LIN {X 0.080,Y -429.880,Z 672.901,A 0.000,B 0.000,C 90.000,E1 18.181} C_DIS
LIN {X -0.115,Y -431.372,Z 672.890,A 0.000,B 0.000,C 90.000,E1 16.205} C_DIS
LIN {X -0.059,Y -433.748,Z 672.875,A 0.000,B 0.000,C 90.000,E1 13.536} C_DIS
LIN {X 0.029,Y -435.804,Z 672.864,A 0.000,B 0.000,C 90.000,E1 11.535} C_DIS
LIN {X 0.134,Y -438.251,Z 672.851,A 0.000,B 0.000,C 90.000,E1 9.208} C_DIS
LIN {X -0.200,Y -440.989,Z 672.839,A 0.000,B 0.000,C 90.000,E1 6.947} C_DIS
LIN {X 0.152,Y -443.481,Z 672.828,A 0.000,B 0.000,C 90.000,E1 4.935} C_DIS
LIN {X -0.046,Y -447.163,Z 672.813,A 0.000,B 0.000,C 90.000,E1 2.350} C_DIS
LIN {X -0.119,Y -451.557,Z 672.797,A 0.000,B 0.000,C 90.000,E1 359.484} C_DIS
LIN {X 0.170,Y -455.546,Z 672.785,A 0.000,B 0.000,C 90.000,E1 357.192} C_DIS
LIN {X 0.214,Y -458.466,Z 672.776,A 0.000,B 0.000,C 90.000,E1 355.584} C_DIS
LIN {X -0.148,Y -461.460,Z 672.767,A 0.000,B 0.000,C 90.000,E1 354.033} C_DIS
LIN {X 0.093,Y -465.598,Z 672.754,A 0.000,B 0.000,C 90.000,E1 351.781} C_DIS
LIN {X -0.140,Y -469.084,Z 672.744,A 0.000,B 0.000,C 90.000,E1 349.916} C_DIS
LIN {X 0.174,Y -472.431,Z 672.733,A 0.000,B 0.000,C 90.000,E1 347.993} C_DIS
LIN {X 0.025,Y -476.365,Z 672.721,A 0.000,B 0.000,C 90.000,E1 345.825} C_DIS
LIN {X -0.099,Y -479.865,Z 672.711,A 0.000,B 0.000,C 90.000,E1 343.976} C_DIS
LIN {X -0.142,Y -483.419,Z 672.701,A 0.000,B 0.000,C 90.000,E1 342.127} C_DIS
LIN {X 0.212,Y -487.775,Z 672.689,A 0.000,B 0.000,C 90.000,E1 339.934} C_DIS
LIN {X 0.229,Y -492.077,Z 672.677,A 0.000,B 0.000,C 90.000,E1 337.794} C_DIS
LIN {X -0.025,Y -494.971,Z 672.668,A 0.000,B 0.000,C 90.000,E1 336.305} C_DIS
LIN {X -0.028,Y -497.759,Z 672.660,A 0.000,B 0.000,C 90.000,E1 334.793} C_DIS
LIN {X 0.240,Y -500.778,Z 672.652,A 0.000,B 0.000,C 90.000,E1 333.256} C_DIS
LIN {X -0.147,Y -501.596,Z 672.650,A 0.000,B 0.000,C 90.000,E1 332.999} C_DIS
LIN {X 0.034,Y -502.535,Z 672.648,A 0.000,B 0.000,C 90.000,E1 332.692} C_DIS
LIN {X -0.118,Y -503.291,Z 672.647,A 0.000,B 0.000,C 90.000,E1 332.410} C_DIS
LIN {X 0.254,Y -505.894,Z 672.643,A 0.000,B 0.000,C 90.000,E1 331.769} C_DIS
LIN {X 0.141,Y -507.043,Z 672.642,A 0.000,B 0.000,C 90.000,E1 331.591} C_DIS
LIN {X 0.151,Y -510.292,Z 672.640,A 0.000,B 0.000,C 90.000,E1 331.179} C_DIS
LIN {X 0.180,Y -513.746,Z 672.638,A 0.000,B 0.000,C 90.000,E1 330.845} C_DIS
LIN {X 0.160,Y -516.813,Z 672.637,A 0.000,B 0.000,C 90.000,E1 330.589} C_DIS
LIN {X 0.046,Y -533.052,Z 672.630,A 0.000,B 0.000,C 90.000,E1 329.459} C_DIS
LIN {X -0.033,Y -540.415,Z 672.627,A 0.000,B 0.000,C 90.000,E1 328.918} C_DIS
LIN {X -0.038,Y -546.271,Z 672.625,A 0.000,B 0.000,C 90.000,E1 328.456} C_DIS
LIN {X -0.173,Y -551.951,Z 672.622,A 0.000,B 0.000,C 90.000,E1 327.995} C_DIS
LIN {X -0.024,Y -560.113,Z 672.618,A 0.000,B 0.000,C 90.000,E1 327.248} C_DIS
LIN {X -0.061,Y -569.208,Z 672.613,A 0.000,B 0.000,C 90.000,E1 326.373} C_DIS
LIN {X -0.056,Y -578.305,Z 672.608,A 0.000,B 0.000,C 90.000,E1 325.468} C_DIS
LIN {X 0.240,Y -588.531,Z 672.602,A 0.000,B 0.000,C 90.000,E1 324.402} C_DIS
LIN {X -0.015,Y -593.457,Z 672.600,A 0.000,B 0.000,C 90.000,E1 323.909} C_DIS
LIN {X 0.212,Y -600.526,Z 672.595,A 0.000,B 0.000,C 90.000,E1 323.130} C_DIS
LIN {X 0.309,Y -606.223,Z 672.592,A 0.000,B 0.000,C 90.000,E1 322.477} C_DIS
LIN {X 0.322,Y -611.798,Z 672.588,A 0.000,B 0.000,C 90.000,E1 321.823} C_DIS
LIN {X -0.183,Y -618.774,Z 672.583,A 0.000,B 0.000,C 90.000,E1 320.964} C_DIS
LIN {X 0.324,Y -623.427,Z 672.580,A 0.000,B 0.000,C 90.000,E1 320.275} C_DIS
LIN {X 0.001,Y -627.856,Z 672.576,A 0.000,B 0.000,C 90.000,E1 319.666} C_DIS
LIN {X -0.318,Y -632.855,Z 672.572,A 0.000,B 0.000,C 90.000,E1 318.933} C_DIS
LIN {X -0.175,Y -637.627,Z 672.568,A 0.000,B 0.000,C 90.000,E1 318.162} C_DIS
LIN {X -0.006,Y -642.937,Z 672.563,A 0.000,B 0.000,C 90.000,E1 317.268} C_DIS
LIN {X -0.301,Y -648.669,Z 672.557,A 0.000,B 0.000,C 90.000,E1 316.296} C_DIS
LIN {X -0.051,Y -654.087,Z 672.552,A 0.000,B 0.000,C 90.000,E1 315.283} C_DIS
LIN {X -0.180,Y -658.514,Z 672.547,A 0.000,B 0.000,C 90.000,E1 314.433} C_DIS
LIN {X 0.187,Y -663.844,Z 672.541,A 0.000,B 0.000,C 90.000,E1 313.299} C_DIS
LIN {X -0.302,Y -668.345,Z 672.535,A 0.000,B 0.000,C 90.000,E1 312.366} C_DIS
LIN {X 0.201,Y -671.663,Z 672.531,A 0.000,B 0.000,C 90.000,E1 311.595} C_DIS
LIN {X -0.103,Y -676.763,Z 672.525,A 0.000,B 0.000,C 90.000,E1 310.415} C_DIS
LIN {X -0.034,Y -679.526,Z 672.521,A 0.000,B 0.000,C 90.000,E1 309.688} C_DIS
LIN {X 0.113,Y -681.274,Z 672.518,A 0.000,B 0.000,C 90.000,E1 309.197} C_DIS
LIN {X -0.041,Y -685.072,Z 672.511,A 0.000,B 0.000,C 90.000,E1 308.016} C_DIS
LIN {X -0.223,Y -687.170,Z 672.507,A 0.000,B 0.000,C 90.000,E1 307.317} C_DIS
LIN {X -0.337,Y -689.640,Z 672.502,A 0.000,B 0.000,C 90.000,E1 306.377} C_DIS
LIN {X 0.137,Y -691.969,Z 672.497,A 0.000,B 0.000,C 90.000,E1 305.391} C_DIS
LIN {X 0.070,Y -694.004,Z 672.491,A 0.000,B 0.000,C 90.000,E1 304.452} C_DIS
LIN {X 0.203,Y -695.870,Z 672.486,A 0.000,B 0.000,C 90.000,E1 303.499} C_DIS
LIN {X 0.366,Y -697.540,Z 672.481,A 0.000,B 0.000,C 90.000,E1 302.546} C_DIS
LIN {X 0.206,Y -699.243,Z 672.474,A 0.000,B 0.000,C 90.000,E1 301.386} C_DIS
LIN {X 0.045,Y -700.466,Z 672.469,A 0.000,B 0.000,C 90.000,E1 300.463} C_DIS
LIN {X -0.097,Y -701.424,Z 672.464,A 0.000,B 0.000,C 90.000,E1 299.539} C_DIS
LIN {X 0.048,Y -702.476,Z 672.458,A 0.000,B 0.000,C 90.000,E1 298.359} C_DIS
LIN {X -0.179,Y -703.813,Z 672.449,A 0.000,B 0.000,C 90.000,E1 296.744} C_DIS
LIN {X 0.021,Y -704.458,Z 672.443,A 0.000,B 0.000,C 90.000,E1 295.796} C_DIS
LIN {X -0.327,Y -704.513,Z 672.442,A 0.000,B 0.000,C 90.000,E1 295.591} C_DIS
LIN {X 0.245,Y -704.053,Z 672.440,A 0.000,B 0.000,C 90.000,E1 295.079} C_DIS
LIN {X -0.406,Y -703.556,Z 672.438,A 0.000,B 0.000,C 90.000,E1 294.899} C_DIS
LIN {X 0.159,Y -701.504,Z 672.436,A 0.000,B 0.000,C 90.000,E1 294.387} C_DIS
LIN {X 0.297,Y -700.902,Z 672.435,A 0.000,B 0.000,C 90.000,E1 294.259} C_DIS
LIN {X 0.148,Y -699.998,Z 672.434,A 0.000,B 0.000,C 90.000,E1 294.155} C_DIS
LIN {X -0.354,Y -698.653,Z 672.434,A 0.000,B 0.000,C 90.000,E1 294.079} C_DIS
LIN {X -0.100,Y -692.661,Z 672.431,A 0.000,B 0.000,C 90.000,E1 293.643} C_DIS
LIN {X 0.271,Y -690.364,Z 672.431,A 0.000,B 0.000,C 90.000,E1 293.515} C_DIS
LIN {X 0.067,Y -688.120,Z 672.430,A 0.000,B 0.000,C 90.000,E1 293.462} C_DIS
LIN {X 0.247,Y -679.913,Z 672.429,A 0.000,B 0.000,C 90.000,E1 293.259} C_DIS
LIN {X 0.214,Y -670.677,Z 672.429,A 0.000,B 0.000,C 90.000,E1 293.153} C_DIS
LIN {X -0.217,Y -665.106,Z 672.428,A 0.000,B 0.000,C 90.000,E1 293.131} C_DIS
LIN {X 0.275,Y -655.083,Z 672.428,A 0.000,B 0.000,C 90.000,E1 292.950} C_DIS
LIN {X -0.154,Y -645.323,Z 672.427,A 0.000,B 0.000,C 90.000,E1 292.823} C_DIS
LIN {X 0.209,Y -635.120,Z 672.426,A 0.000,B 0.000,C 90.000,E1 292.589} C_DIS
LIN {X 0.133,Y -621.781,Z 672.424,A 0.000,B 0.000,C 90.000,E1 292.280} C_DIS
LIN {X -0.232,Y -604.948,Z 672.421,A 0.000,B 0.000,C 90.000,E1 291.844} C_DIS
LIN {X -0.161,Y -577.296,Z 672.416,A 0.000,B 0.000,C 90.000,E1 290.972} C_DIS
LIN {X -0.053,Y -563.094,Z 672.414,A 0.000,B 0.000,C 90.000,E1 290.556} C_DIS
LIN {X -0.047,Y -556.572,Z 672.413,A 0.000,B 0.000,C 90.000,E1 290.248} C_DIS
LIN {X -0.095,Y -556.479,Z 672.412,A 0.000,B 0.000,C 90.000,E1 290.248} C_DIS
LIN {X 0.094,Y -555.287,Z 672.412,A 0.000,B 0.000,C 90.000,E1 290.066} C_DIS
LIN {X 0.052,Y -555.271,Z 672.412,A 0.000,B 0.000,C 90.000,E1 290.066} C_DIS
LIN {X 0.022,Y -554.576,Z 672.410,A 0.000,B 0.000,C 90.000,E1 289.704} C_DIS
LIN {X 0.188,Y -554.054,Z 672.399,A 0.000,B 0.000,C 90.000,E1 287.873} C_DIS
LIN {X -0.264,Y -553.758,Z 672.393,A 0.000,B 0.000,C 90.000,E1 286.804} C_DIS
LIN {X -0.328,Y -553.213,Z 672.384,A 0.000,B 0.000,C 90.000,E1 285.134} C_DIS
LIN {X 0.001,Y -552.630,Z 672.376,A 0.000,B 0.000,C 90.000,E1 283.703} C_DIS
LIN {X 0.054,Y -551.874,Z 672.368,A 0.000,B 0.000,C 90.000,E1 282.299} C_DIS
LIN {X 0.215,Y -551.004,Z 672.359,A 0.000,B 0.000,C 90.000,E1 280.602} C_DIS
LIN {X -0.182,Y -550.230,Z 672.348,A 0.000,B 0.000,C 90.000,E1 278.681} C_DIS
LIN {X 0.195,Y -549.869,Z 672.340,A 0.000,B 0.000,C 90.000,E1 277.239} C_DIS
LIN {X 0.024,Y -549.613,Z 672.333,A 0.000,B 0.000,C 90.000,E1 275.853} C_DIS
LIN {X -0.029,Y -549.376,Z 672.320,A 0.000,B 0.000,C 90.000,E1 273.612} C_DIS
LIN {X 0.252,Y -549.149,Z 672.312,A 0.000,B 0.000,C 90.000,E1 272.178} C_DIS
LIN {X -0.074,Y -548.777,Z 672.306,A 0.000,B 0.000,C 90.000,E1 271.088} C_DIS
LIN {X 0.180,Y -548.088,Z 672.298,A 0.000,B 0.000,C 90.000,E1 269.656} C_DIS
LIN {X -0.130,Y -547.287,Z 672.290,A 0.000,B 0.000,C 90.000,E1 268.282} C_DIS
LIN {X 0.173,Y -546.280,Z 672.281,A 0.000,B 0.000,C 90.000,E1 266.560} C_DIS
LIN {X -0.115,Y -545.287,Z 672.273,A 0.000,B 0.000,C 90.000,E1 265.179} C_DIS
LIN {X 0.120,Y -544.116,Z 672.265,A 0.000,B 0.000,C 90.000,E1 263.742} C_DIS
LIN {X -0.232,Y -543.078,Z 672.259,A 0.000,B 0.000,C 90.000,E1 262.648} C_DIS
LIN {X 0.163,Y -541.204,Z 672.250,A 0.000,B 0.000,C 90.000,E1 260.905} C_DIS
LIN {X 0.140,Y -539.088,Z 672.237,A 0.000,B 0.000,C 90.000,E1 258.634} C_DIS
LIN {X 0.209,Y -536.968,Z 672.223,A 0.000,B 0.000,C 90.000,E1 256.061} C_DIS
LIN {X 0.240,Y -535.696,Z 672.215,A 0.000,B 0.000,C 90.000,E1 254.629} C_DIS
LIN {X 0.063,Y -534.559,Z 672.208,A 0.000,B 0.000,C 90.000,E1 253.504} C_DIS
LIN {X -0.044,Y -532.250,Z 672.196,A 0.000,B 0.000,C 90.000,E1 251.221} C_DIS
LIN {X -0.143,Y -531.429,Z 672.191,A 0.000,B 0.000,C 90.000,E1 250.369} C_DIS
LIN {X -0.061,Y -529.990,Z 672.185,A 0.000,B 0.000,C 90.000,E1 249.209} C_DIS
LIN {X -0.133,Y -527.570,Z 672.175,A 0.000,B 0.000,C 90.000,E1 247.486} C_DIS
LIN {X 0.084,Y -525.904,Z 672.168,A 0.000,B 0.000,C 90.000,E1 246.305} C_DIS
LIN {X -0.141,Y -522.911,Z 672.159,A 0.000,B 0.000,C 90.000,E1 244.588} C_DIS
LIN {X 0.222,Y -520.768,Z 672.152,A 0.000,B 0.000,C 90.000,E1 243.384} C_DIS
LIN {X 0.119,Y -517.300,Z 672.143,A 0.000,B 0.000,C 90.000,E1 241.641} C_DIS
LIN {X 0.171,Y -514.866,Z 672.136,A 0.000,B 0.000,C 90.000,E1 240.461} C_DIS
LIN {X 0.090,Y -511.648,Z 672.128,A 0.000,B 0.000,C 90.000,E1 238.997} C_DIS
LIN {X -0.052,Y -508.421,Z 672.120,A 0.000,B 0.000,C 90.000,E1 237.533} C_DIS
LIN {X 0.289,Y -505.035,Z 672.111,A 0.000,B 0.000,C 90.000,E1 236.008} C_DIS
LIN {X -0.019,Y -502.131,Z 672.105,A 0.000,B 0.000,C 90.000,E1 234.848} C_DIS
LIN {X -0.039,Y -497.638,Z 672.095,A 0.000,B 0.000,C 90.000,E1 233.050} C_DIS
LIN {X 0.010,Y -492.473,Z 672.083,A 0.000,B 0.000,C 90.000,E1 230.928} C_DIS
LIN {X 0.091,Y -489.603,Z 672.076,A 0.000,B 0.000,C 90.000,E1 229.703} C_DIS
LIN {X 0.210,Y -485.948,Z 672.068,A 0.000,B 0.000,C 90.000,E1 228.162} C_DIS
LIN {X -0.026,Y -480.144,Z 672.054,A 0.000,B 0.000,C 90.000,E1 225.729} C_DIS
LIN {X 0.013,Y -475.706,Z 672.044,A 0.000,B 0.000,C 90.000,E1 223.866} C_DIS
LIN {X -0.031,Y -471.424,Z 672.033,A 0.000,B 0.000,C 90.000,E1 222.000} C_DIS
LIN {X 0.002,Y -466.055,Z 672.019,A 0.000,B 0.000,C 90.000,E1 219.483} C_DIS
LIN {X 0.101,Y -462.792,Z 672.011,A 0.000,B 0.000,C 90.000,E1 217.890} C_DIS
LIN {X -0.009,Y -458.282,Z 671.998,A 0.000,B 0.000,C 90.000,E1 215.678} C_DIS
LIN {X -0.230,Y -454.694,Z 671.988,A 0.000,B 0.000,C 90.000,E1 213.785} C_DIS
LIN {X 0.213,Y -451.026,Z 671.977,A 0.000,B 0.000,C 90.000,E1 211.799} C_DIS
LIN {X 0.167,Y -446.761,Z 671.964,A 0.000,B 0.000,C 90.000,E1 209.539} C_DIS
LIN {X 0.176,Y -442.726,Z 671.952,A 0.000,B 0.000,C 90.000,E1 207.257} C_DIS
LIN {X -0.010,Y -439.755,Z 671.943,A 0.000,B 0.000,C 90.000,E1 205.643} C_DIS
LIN {X 0.017,Y -435.666,Z 671.930,A 0.000,B 0.000,C 90.000,E1 203.334} C_DIS
LIN {X -0.047,Y -432.011,Z 671.919,A 0.000,B 0.000,C 90.000,E1 201.354} C_DIS
LIN {X 0.196,Y -428.409,Z 671.908,A 0.000,B 0.000,C 90.000,E1 199.322} C_DIS
LIN {X -0.090,Y -423.799,Z 671.893,A 0.000,B 0.000,C 90.000,E1 196.677} C_DIS
LIN {X 0.180,Y -420.959,Z 671.883,A 0.000,B 0.000,C 90.000,E1 194.954} C_DIS
LIN {X -0.178,Y -418.673,Z 671.876,A 0.000,B 0.000,C 90.000,E1 193.647} C_DIS
LIN {X 0.068,Y -413.636,Z 671.859,A 0.000,B 0.000,C 90.000,E1 190.546} C_DIS
LIN {X -0.136,Y -411.008,Z 671.849,A 0.000,B 0.000,C 90.000,E1 188.859} C_DIS
LIN {X -0.028,Y -407.872,Z 671.838,A 0.000,B 0.000,C 90.000,E1 186.777} C_DIS
LIN {X -0.120,Y -403.635,Z 671.820,A 0.000,B 0.000,C 90.000,E1 183.669} C_DIS
LIN {X 0.094,Y -401.103,Z 671.809,A 0.000,B 0.000,C 90.000,E1 181.547} C_DIS
LIN {X 0.125,Y -398.349,Z 671.793,A 0.000,B 0.000,C 90.000,E1 178.740} C_DIS
LIN {X -0.061,Y -395.440,Z 671.772,A 0.000,B 0.000,C 90.000,E1 174.894} C_DIS
LIN {X -0.008,Y -394.198,Z 671.758,A 0.000,B 0.000,C 90.000,E1 172.413} C_DIS
LIN {X 0.097,Y -393.498,Z 671.746,A 0.000,B 0.000,C 90.000,E1 170.274} C_DIS
LIN {X -0.076,Y -393.038,Z 671.734,A 0.000,B 0.000,C 90.000,E1 168.173} C_DIS
LIN {X -0.083,Y -392.879,Z 671.722,A 0.000,B 0.000,C 90.000,E1 166.047} C_DIS
LIN {X 0.010,Y -392.836,Z 671.707,A 0.000,B 0.000,C 90.000,E1 163.196} C_DIS
LIN {X -0.109,Y -392.982,Z 671.693,A 0.000,B 0.000,C 90.000,E1 160.732} C_DIS
LIN {X -0.078,Y -393.142,Z 671.683,A 0.000,B 0.000,C 90.000,E1 158.954} C_DIS
LIN {X 0.155,Y -393.420,Z 671.671,A 0.000,B 0.000,C 90.000,E1 156.794} C_DIS
LIN {X -0.175,Y -393.732,Z 671.659,A 0.000,B 0.000,C 90.000,E1 154.717} C_DIS
LIN {X 0.018,Y -394.135,Z 671.648,A 0.000,B 0.000,C 90.000,E1 152.564} C_DIS
LIN {X 0.018,Y -394.563,Z 671.638,A 0.000,B 0.000,C 90.000,E1 150.795} C_DIS
LIN {X 0.227,Y -394.992,Z 671.628,A 0.000,B 0.000,C 90.000,E1 148.997} C_DIS
LIN {X -0.024,Y -395.679,Z 671.616,A 0.000,B 0.000,C 90.000,E1 146.914} C_DIS
LIN {X 0.227,Y -397.116,Z 671.599,A 0.000,B 0.000,C 90.000,E1 143.703} C_DIS
LIN {X -0.050,Y -398.754,Z 671.583,A 0.000,B 0.000,C 90.000,E1 140.928} C_DIS
LIN {X -0.142,Y -400.412,Z 671.569,A 0.000,B 0.000,C 90.000,E1 138.485} C_DIS
LIN {X -0.018,Y -401.423,Z 671.562,A 0.000,B 0.000,C 90.000,E1 137.067} C_DIS
LIN {X -0.222,Y -402.976,Z 671.550,A 0.000,B 0.000,C 90.000,E1 135.000} C_DIS
LIN {X -0.172,Y -404.024,Z 671.544,A 0.000,B 0.000,C 90.000,E1 133.947} C_DIS
LIN {X -0.050,Y -404.439,Z 671.542,A 0.000,B 0.000,C 90.000,E1 133.581} C_DIS
LIN {X 0.102,Y -406.028,Z 671.537,A 0.000,B 0.000,C 90.000,E1 132.690} C_DIS
LIN {X 0.018,Y -406.708,Z 671.536,A 0.000,B 0.000,C 90.000,E1 132.528} C_DIS
LIN {X 0.114,Y -408.061,Z 671.534,A 0.000,B 0.000,C 90.000,E1 132.081} C_DIS
LIN {X -0.167,Y -411.535,Z 671.531,A 0.000,B 0.000,C 90.000,E1 131.515} C_DIS
LIN {X -0.159,Y -415.629,Z 671.528,A 0.000,B 0.000,C 90.000,E1 131.067} C_DIS
LIN {X 0.221,Y -419.960,Z 671.526,A 0.000,B 0.000,C 90.000,E1 130.620} C_DIS
LIN {X 0.233,Y -426.338,Z 671.523,A 0.000,B 0.000,C 90.000,E1 130.092} C_DIS
LIN {X -0.083,Y -438.989,Z 671.517,A 0.000,B 0.000,C 90.000,E1 129.116} C_DIS
LIN {X -0.280,Y -451.694,Z 671.512,A 0.000,B 0.000,C 90.000,E1 128.177} C_DIS
LIN {X -0.085,Y -462.693,Z 671.507,A 0.000,B 0.000,C 90.000,E1 127.317} C_DIS
LIN {X 0.259,Y -468.883,Z 671.505,A 0.000,B 0.000,C 90.000,E1 126.790} C_DIS
LIN {X 0.223,Y -474.927,Z 671.502,A 0.000,B 0.000,C 90.000,E1 126.297} C_DIS
LIN {X -0.306,Y -483.884,Z 671.498,A 0.000,B 0.000,C 90.000,E1 125.598} C_DIS
LIN {X 0.325,Y -489.478,Z 671.495,A 0.000,B 0.000,C 90.000,E1 125.025} C_DIS
LIN {X -0.058,Y -498.082,Z 671.490,A 0.000,B 0.000,C 90.000,E1 124.278} C_DIS
LIN {X 0.218,Y -507.801,Z 671.485,A 0.000,B 0.000,C 90.000,E1 123.293} C_DIS
LIN {X 0.159,Y -513.178,Z 671.482,A 0.000,B 0.000,C 90.000,E1 122.752} C_DIS
LIN {X 0.098,Y -517.122,Z 671.480,A 0.000,B 0.000,C 90.000,E1 122.339} C_DIS
LIN {X -0.191,Y -524.458,Z 671.475,A 0.000,B 0.000,C 90.000,E1 121.544} C_DIS
LIN {X -0.068,Y -530.842,Z 671.471,A 0.000,B 0.000,C 90.000,E1 120.747} C_DIS
LIN {X -0.213,Y -534.927,Z 671.468,A 0.000,B 0.000,C 90.000,E1 120.207} C_DIS
LIN {X -0.148,Y -538.528,Z 671.465,A 0.000,B 0.000,C 90.000,E1 119.667} C_DIS
LIN {X 0.013,Y -542.761,Z 671.461,A 0.000,B 0.000,C 90.000,E1 118.949} C_DIS
LIN {X 0.106,Y -546.658,Z 671.457,A 0.000,B 0.000,C 90.000,E1 118.231} C_DIS
LIN {X 0.117,Y -550.807,Z 671.452,A 0.000,B 0.000,C 90.000,E1 117.385} C_DIS
LIN {X 0.058,Y -555.180,Z 671.447,A 0.000,B 0.000,C 90.000,E1 116.411} C_DIS
LIN {X 0.226,Y -557.009,Z 671.445,A 0.000,B 0.000,C 90.000,E1 115.976} C_DIS
LIN {X 0.095,Y -560.371,Z 671.440,A 0.000,B 0.000,C 90.000,E1 115.155} C_DIS
LIN {X -0.200,Y -564.406,Z 671.434,A 0.000,B 0.000,C 90.000,E1 114.079} C_DIS
LIN {X 0.259,Y -567.071,Z 671.429,A 0.000,B 0.000,C 90.000,E1 113.206} C_DIS
LIN {X 0.009,Y -569.520,Z 671.425,A 0.000,B 0.000,C 90.000,E1 112.408} C_DIS
LIN {X -0.181,Y -572.296,Z 671.418,A 0.000,B 0.000,C 90.000,E1 111.334} C_DIS
LIN {X 0.154,Y -574.143,Z 671.414,A 0.000,B 0.000,C 90.000,E1 110.482} C_DIS
LIN {X -0.023,Y -576.962,Z 671.406,A 0.000,B 0.000,C 90.000,E1 109.141} C_DIS
LIN {X 0.041,Y -580.202,Z 671.397,A 0.000,B 0.000,C 90.000,E1 107.511} C_DIS
LIN {X 0.172,Y -582.899,Z 671.390,A 0.000,B 0.000,C 90.000,E1 106.150} C_DIS
LIN {X 0.282,Y -584.983,Z 671.384,A 0.000,B 0.000,C 90.000,E1 105.064} C_DIS
LIN {X 0.043,Y -587.985,Z 671.375,A 0.000,B 0.000,C 90.000,E1 103.480} C_DIS
LIN {X 0.001,Y -590.947,Z 671.366,A 0.000,B 0.000,C 90.000,E1 101.883} C_DIS
LIN {X 0.319,Y -594.814,Z 671.354,A 0.000,B 0.000,C 90.000,E1 99.726} C_DIS
LIN {X 0.065,Y -597.545,Z 671.345,A 0.000,B 0.000,C 90.000,E1 98.163} C_DIS
LIN {X 0.167,Y -599.558,Z 671.338,A 0.000,B 0.000,C 90.000,E1 96.834} C_DIS
LIN {X 0.240,Y -601.526,Z 671.331,A 0.000,B 0.000,C 90.000,E1 95.511} C_DIS
LIN {X 0.105,Y -602.986,Z 671.325,A 0.000,B 0.000,C 90.000,E1 94.473} C_DIS
LIN {X 0.196,Y -604.621,Z 671.318,A 0.000,B 0.000,C 90.000,E1 93.154} C_DIS
LIN {X -0.284,Y -606.004,Z 671.310,A 0.000,B 0.000,C 90.000,E1 91.892} C_DIS
LIN {X 0.194,Y -606.931,Z 671.305,A 0.000,B 0.000,C 90.000,E1 90.802} C_DIS
LIN {X -0.271,Y -607.800,Z 671.297,A 0.000,B 0.000,C 90.000,E1 89.542} C_DIS
LIN {X -0.059,Y -608.120,Z 671.293,A 0.000,B 0.000,C 90.000,E1 88.740} C_DIS
LIN {X -0.220,Y -608.607,Z 671.284,A 0.000,B 0.000,C 90.000,E1 87.192} C_DIS
LIN {X -0.001,Y -608.743,Z 671.277,A 0.000,B 0.000,C 90.000,E1 85.869} C_DIS
LIN {X 0.172,Y -608.576,Z 671.270,A 0.000,B 0.000,C 90.000,E1 84.552} C_DIS
LIN {X 0.126,Y -608.333,Z 671.264,A 0.000,B 0.000,C 90.000,E1 83.514} C_DIS
LIN {X -0.201,Y -607.803,Z 671.257,A 0.000,B 0.000,C 90.000,E1 82.243} C_DIS
LIN {X -0.171,Y -607.189,Z 671.251,A 0.000,B 0.000,C 90.000,E1 81.197} C_DIS
LIN {X 0.123,Y -606.498,Z 671.247,A 0.000,B 0.000,C 90.000,E1 80.387} C_DIS
LIN {X 0.188,Y -604.896,Z 671.238,A 0.000,B 0.000,C 90.000,E1 78.814} C_DIS
LIN {X 0.023,Y -603.344,Z 671.231,A 0.000,B 0.000,C 90.000,E1 77.521} C_DIS
LIN {X 0.110,Y -601.986,Z 671.225,A 0.000,B 0.000,C 90.000,E1 76.464} C_DIS
LIN {X 0.171,Y -600.532,Z 671.219,A 0.000,B 0.000,C 90.000,E1 75.408} C_DIS
LIN {X -0.218,Y -598.977,Z 671.213,A 0.000,B 0.000,C 90.000,E1 74.393} C_DIS
LIN {X -0.342,Y -596.879,Z 671.206,A 0.000,B 0.000,C 90.000,E1 73.087} C_DIS
LIN {X -0.032,Y -595.042,Z 671.200,A 0.000,B 0.000,C 90.000,E1 72.000} C_DIS
LIN {X -0.056,Y -592.639,Z 671.193,A 0.000,B 0.000,C 90.000,E1 70.678} C_DIS
LIN {X 0.067,Y -589.912,Z 671.185,A 0.000,B 0.000,C 90.000,E1 69.337} C_DIS
LIN {X -0.072,Y -587.441,Z 671.179,A 0.000,B 0.000,C 90.000,E1 68.284} C_DIS
LIN {X -0.114,Y -585.354,Z 671.175,A 0.000,B 0.000,C 90.000,E1 67.486} C_DIS
LIN {X -0.081,Y -582.283,Z 671.169,A 0.000,B 0.000,C 90.000,E1 66.410} C_DIS
LIN {X -0.322,Y -578.843,Z 671.163,A 0.000,B 0.000,C 90.000,E1 65.357} C_DIS
LIN {X -0.226,Y -576.069,Z 671.158,A 0.000,B 0.000,C 90.000,E1 64.537} C_DIS
LIN {X -0.065,Y -572.029,Z 671.152,A 0.000,B 0.000,C 90.000,E1 63.435} C_DIS
LIN {X 0.122,Y -569.937,Z 671.149,A 0.000,B 0.000,C 90.000,E1 62.871} C_DIS
LIN {X 0.286,Y -565.907,Z 671.144,A 0.000,B 0.000,C 90.000,E1 61.897} C_DIS
LIN {X -0.001,Y -562.131,Z 671.140,A 0.000,B 0.000,C 90.000,E1 61.101} C_DIS
LIN {X 0.094,Y -559.437,Z 671.136,A 0.000,B 0.000,C 90.000,E1 60.539} C_DIS
LIN {X -0.085,Y -555.571,Z 671.133,A 0.000,B 0.000,C 90.000,E1 59.871} C_DIS
LIN {X 0.111,Y -551.144,Z 671.129,A 0.000,B 0.000,C 90.000,E1 59.154} C_DIS
LIN {X -0.083,Y -547.307,Z 671.126,A 0.000,B 0.000,C 90.000,E1 58.614} C_DIS
LIN {X -0.012,Y -543.185,Z 671.122,A 0.000,B 0.000,C 90.000,E1 58.043} C_DIS
LIN {X 0.200,Y -538.534,Z 671.119,A 0.000,B 0.000,C 90.000,E1 57.454} C_DIS
LIN {X 0.014,Y -533.355,Z 671.116,A 0.000,B 0.000,C 90.000,E1 56.914} C_DIS
LIN {X 0.065,Y -529.630,Z 671.114,A 0.000,B 0.000,C 90.000,E1 56.548} C_DIS
LIN {X -0.144,Y -524.075,Z 671.112,A 0.000,B 0.000,C 90.000,E1 56.087} C_DIS
LIN {X 0.227,Y -518.081,Z 671.109,A 0.000,B 0.000,C 90.000,E1 55.595} C_DIS
LIN {X 0.174,Y -513.201,Z 671.107,A 0.000,B 0.000,C 90.000,E1 55.261} C_DIS
LIN {X 0.022,Y -504.900,Z 671.104,A 0.000,B 0.000,C 90.000,E1 54.769} C_DIS
LIN {X 0.220,Y -496.773,Z 671.102,A 0.000,B 0.000,C 90.000,E1 54.276} C_DIS
LIN {X -0.247,Y -480.054,Z 671.097,A 0.000,B 0.000,C 90.000,E1 53.417} C_DIS
LIN {X -0.023,Y -463.539,Z 671.092,A 0.000,B 0.000,C 90.000,E1 52.477} C_DIS
LIN {X -0.068,Y -442.276,Z 671.085,A 0.000,B 0.000,C 90.000,E1 51.251} C_DIS
LIN {X 0.026,Y -430.772,Z 671.081,A 0.000,B 0.000,C 90.000,E1 50.517} C_DIS
LIN {X 0.004,Y -430.761,Z 671.081,A 0.000,B 0.000,C 90.000,E1 50.517} C_DIS
LIN {X -0.049,Y -421.534,Z 671.058,A 0.000,B 0.000,C 90.000,E1 46.419} C_DIS
LIN {X 0.017,Y -418.402,Z 671.048,A 0.000,B 0.000,C 90.000,E1 44.717} C_DIS
LIN {X 0.054,Y -416.550,Z 671.044,A 0.000,B 0.000,C 90.000,E1 43.947} C_DIS
LIN {X -0.036,Y -416.455,Z 671.043,A 0.000,B 0.000,C 90.000,E1 43.704} C_DIS
LIN {X -0.050,Y -416.490,Z 671.033,A 0.000,B 0.000,C 90.000,E1 42.000} C_DIS
LIN {X -0.280,Y -416.815,Z 671.020,A 0.000,B 0.000,C 90.000,E1 39.644} C_DIS
LIN {X -0.134,Y -418.067,Z 671.001,A 0.000,B 0.000,C 90.000,E1 36.217} C_DIS
LIN {X 0.141,Y -418.796,Z 670.994,A 0.000,B 0.000,C 90.000,E1 34.818} C_DIS
LIN {X -0.048,Y -419.976,Z 670.980,A 0.000,B 0.000,C 90.000,E1 32.467} C_DIS
LIN {X -0.235,Y -420.926,Z 670.971,A 0.000,B 0.000,C 90.000,E1 30.797} C_DIS
LIN {X -0.037,Y -421.818,Z 670.962,A 0.000,B 0.000,C 90.000,E1 29.077} C_DIS
LIN {X -0.026,Y -422.815,Z 670.952,A 0.000,B 0.000,C 90.000,E1 27.385} C_DIS
LIN {X -0.190,Y -423.920,Z 670.943,A 0.000,B 0.000,C 90.000,E1 25.720} C_DIS
LIN {X -0.048,Y -427.375,Z 670.920,A 0.000,B 0.000,C 90.000,E1 21.663} C_DIS
LIN {X -0.086,Y -428.918,Z 670.911,A 0.000,B 0.000,C 90.000,E1 19.993} C_DIS
LIN {X 0.135,Y -429.744,Z 670.905,A 0.000,B 0.000,C 90.000,E1 18.960} C_DIS
LIN {X 0.038,Y -430.743,Z 670.898,A 0.000,B 0.000,C 90.000,E1 17.638} C_DIS
LIN {X 0.077,Y -432.497,Z 670.885,A 0.000,B 0.000,C 90.000,E1 15.300} C_DIS
LIN {X 0.131,Y -434.312,Z 670.874,A 0.000,B 0.000,C 90.000,E1 13.300} C_DIS
LIN {X 0.231,Y -436.337,Z 670.863,A 0.000,B 0.000,C 90.000,E1 11.299} C_DIS
LIN {X -0.087,Y -438.789,Z 670.850,A 0.000,B 0.000,C 90.000,E1 9.029} C_DIS
LIN {X 0.123,Y -441.924,Z 670.836,A 0.000,B 0.000,C 90.000,E1 6.372} C_DIS
LIN {X 0.185,Y -444.868,Z 670.823,A 0.000,B 0.000,C 90.000,E1 4.073} C_DIS
LIN {X 0.023,Y -447.209,Z 670.814,A 0.000,B 0.000,C 90.000,E1 2.465} C_DIS
LIN {X 0.171,Y -451.214,Z 670.799,A 0.000,B 0.000,C 90.000,E1 359.771} C_DIS
LIN {X 0.000,Y -455.139,Z 670.786,A 0.000,B 0.000,C 90.000,E1 357.535} C_DIS
LIN {X 0.222,Y -458.604,Z 670.776,A 0.000,B 0.000,C 90.000,E1 355.584} C_DIS
LIN {X -0.137,Y -461.585,Z 670.767,A 0.000,B 0.000,C 90.000,E1 354.033} C_DIS
LIN {X 0.109,Y -465.712,Z 670.754,A 0.000,B 0.000,C 90.000,E1 351.781} C_DIS
LIN {X 0.063,Y -468.593,Z 670.746,A 0.000,B 0.000,C 90.000,E1 350.208} C_DIS
LIN {X 0.081,Y -471.407,Z 670.737,A 0.000,B 0.000,C 90.000,E1 348.634} C_DIS
LIN {X 0.142,Y -474.174,Z 670.728,A 0.000,B 0.000,C 90.000,E1 347.061} C_DIS
LIN {X 0.004,Y -477.030,Z 670.720,A 0.000,B 0.000,C 90.000,E1 345.519} C_DIS
LIN {X -0.230,Y -480.545,Z 670.709,A 0.000,B 0.000,C 90.000,E1 343.685} C_DIS
LIN {X -0.115,Y -484.710,Z 670.697,A 0.000,B 0.000,C 90.000,E1 341.511} C_DIS
LIN {X 0.093,Y -488.447,Z 670.687,A 0.000,B 0.000,C 90.000,E1 339.645} C_DIS
LIN {X -0.195,Y -492.156,Z 670.677,A 0.000,B 0.000,C 90.000,E1 337.847} C_DIS
LIN {X 0.009,Y -495.030,Z 670.668,A 0.000,B 0.000,C 90.000,E1 336.305} C_DIS
LIN {X 0.008,Y -497.794,Z 670.660,A 0.000,B 0.000,C 90.000,E1 334.793} C_DIS
LIN {X -0.112,Y -501.373,Z 670.650,A 0.000,B 0.000,C 90.000,E1 332.999} C_DIS
LIN {X -0.146,Y -502.900,Z 670.647,A 0.000,B 0.000,C 90.000,E1 332.410} C_DIS
LIN {X -0.035,Y -504.587,Z 670.644,A 0.000,B 0.000,C 90.000,E1 331.948} C_DIS
LIN {X 0.222,Y -505.131,Z 670.643,A 0.000,B 0.000,C 90.000,E1 331.769} C_DIS
LIN {X 0.150,Y -507.629,Z 670.641,A 0.000,B 0.000,C 90.000,E1 331.307} C_DIS
LIN {X -0.035,Y -508.545,Z 670.640,A 0.000,B 0.000,C 90.000,E1 331.179} C_DIS
LIN {X 0.236,Y -511.469,Z 670.638,A 0.000,B 0.000,C 90.000,E1 330.795} C_DIS
LIN {X 0.085,Y -515.255,Z 670.636,A 0.000,B 0.000,C 90.000,E1 330.461} C_DIS
LIN {X -0.098,Y -519.832,Z 670.634,A 0.000,B 0.000,C 90.000,E1 330.127} C_DIS
LIN {X -0.046,Y -532.242,Z 670.629,A 0.000,B 0.000,C 90.000,E1 329.253} C_DIS
LIN {X -0.011,Y -541.183,Z 670.625,A 0.000,B 0.000,C 90.000,E1 328.584} C_DIS
LIN {X 0.053,Y -548.390,Z 670.622,A 0.000,B 0.000,C 90.000,E1 327.995} C_DIS
LIN {X -0.195,Y -558.180,Z 670.618,A 0.000,B 0.000,C 90.000,E1 327.168} C_DIS
LIN {X 0.168,Y -566.112,Z 670.613,A 0.000,B 0.000,C 90.000,E1 326.373} C_DIS
LIN {X -0.270,Y -576.647,Z 670.608,A 0.000,B 0.000,C 90.000,E1 325.388} C_DIS
LIN {X 0.081,Y -586.911,Z 670.602,A 0.000,B 0.000,C 90.000,E1 324.322} C_DIS
LIN {X 0.110,Y -594.401,Z 670.598,A 0.000,B 0.000,C 90.000,E1 323.543} C_DIS
LIN {X -0.248,Y -600.513,Z 670.594,A 0.000,B 0.000,C 90.000,E1 322.924} C_DIS
LIN {X -0.285,Y -606.363,Z 670.590,A 0.000,B 0.000,C 90.000,E1 322.271} C_DIS
LIN {X -0.228,Y -610.872,Z 670.587,A 0.000,B 0.000,C 90.000,E1 321.743} C_DIS
LIN {X 0.122,Y -617.952,Z 670.582,A 0.000,B 0.000,C 90.000,E1 320.803} C_DIS
LIN {X -0.289,Y -623.627,Z 670.578,A 0.000,B 0.000,C 90.000,E1 320.070} C_DIS
LIN {X -0.243,Y -628.879,Z 670.574,A 0.000,B 0.000,C 90.000,E1 319.299} C_DIS
LIN {X -0.169,Y -634.698,Z 670.569,A 0.000,B 0.000,C 90.000,E1 318.405} C_DIS
LIN {X -0.100,Y -640.927,Z 670.563,A 0.000,B 0.000,C 90.000,E1 317.391} C_DIS
LIN {X 0.054,Y -646.798,Z 670.558,A 0.000,B 0.000,C 90.000,E1 316.377} C_DIS
LIN {X 0.255,Y -653.002,Z 670.552,A 0.000,B 0.000,C 90.000,E1 315.243} C_DIS
LIN {X -0.314,Y -656.279,Z 670.548,A 0.000,B 0.000,C 90.000,E1 314.676} C_DIS
LIN {X -0.381,Y -658.811,Z 670.545,A 0.000,B 0.000,C 90.000,E1 314.190} C_DIS
LIN {X 0.010,Y -663.599,Z 670.540,A 0.000,B 0.000,C 90.000,E1 313.176} C_DIS
LIN {X -0.023,Y -668.138,Z 670.534,A 0.000,B 0.000,C 90.000,E1 312.204} C_DIS
LIN {X 0.034,Y -671.476,Z 670.530,A 0.000,B 0.000,C 90.000,E1 311.472} C_DIS
LIN {X 0.064,Y -674.610,Z 670.526,A 0.000,B 0.000,C 90.000,E1 310.744} C_DIS
LIN {X -0.221,Y -678.516,Z 670.521,A 0.000,B 0.000,C 90.000,E1 309.806} C_DIS
LIN {X -0.046,Y -681.110,Z 670.517,A 0.000,B 0.000,C 90.000,E1 309.072} C_DIS
LIN {X 0.191,Y -684.203,Z 670.512,A 0.000,B 0.000,C 90.000,E1 308.096} C_DIS
LIN {X 0.039,Y -687.048,Z 670.506,A 0.000,B 0.000,C 90.000,E1 307.156} C_DIS
LIN {X 0.110,Y -690.162,Z 670.500,A 0.000,B 0.000,C 90.000,E1 305.964} C_DIS
LIN {X 0.028,Y -692.420,Z 670.495,A 0.000,B 0.000,C 90.000,E1 305.025} C_DIS
LIN {X 0.143,Y -694.424,Z 670.489,A 0.000,B 0.000,C 90.000,E1 304.072} C_DIS
LIN {X -0.290,Y -696.284,Z 670.484,A 0.000,B 0.000,C 90.000,E1 303.166} C_DIS
LIN {X -0.120,Y -697.894,Z 670.479,A 0.000,B 0.000,C 90.000,E1 302.212} C_DIS
LIN {X 0.324,Y -699.637,Z 670.472,A 0.000,B 0.000,C 90.000,E1 301.003} C_DIS
LIN {X 0.174,Y -700.801,Z 670.467,A 0.000,B 0.000,C 90.000,E1 300.079} C_DIS
LIN {X -0.298,Y -701.975,Z 670.461,A 0.000,B 0.000,C 90.000,E1 298.949} C_DIS
LIN {X -0.147,Y -702.991,Z 670.454,A 0.000,B 0.000,C 90.000,E1 297.769} C_DIS
LIN {X -0.309,Y -703.994,Z 670.448,A 0.000,B 0.000,C 90.000,E1 296.616} C_DIS
LIN {X -0.106,Y -704.628,Z 670.443,A 0.000,B 0.000,C 90.000,E1 295.668} C_DIS
LIN {X -0.168,Y -704.206,Z 670.440,A 0.000,B 0.000,C 90.000,E1 295.207} C_DIS
LIN {X 0.118,Y -703.903,Z 670.439,A 0.000,B 0.000,C 90.000,E1 294.951} C_DIS
LIN {X -0.249,Y -701.913,Z 670.436,A 0.000,B 0.000,C 90.000,E1 294.515} C_DIS
LIN {X 0.030,Y -700.688,Z 670.435,A 0.000,B 0.000,C 90.000,E1 294.259} C_DIS
LIN {X 0.166,Y -699.707,Z 670.434,A 0.000,B 0.000,C 90.000,E1 294.131} C_DIS
LIN {X 0.018,Y -698.244,Z 670.434,A 0.000,B 0.000,C 90.000,E1 294.027} C_DIS
LIN {X 0.305,Y -693.771,Z 670.432,A 0.000,B 0.000,C 90.000,E1 293.695} C_DIS
LIN {X -0.232,Y -692.221,Z 670.431,A 0.000,B 0.000,C 90.000,E1 293.643} C_DIS
LIN {X 0.202,Y -689.847,Z 670.431,A 0.000,B 0.000,C 90.000,E1 293.515} C_DIS
LIN {X 0.083,Y -684.259,Z 670.430,A 0.000,B 0.000,C 90.000,E1 293.387} C_DIS
LIN {X -0.310,Y -680.456,Z 670.430,A 0.000,B 0.000,C 90.000,E1 293.334} C_DIS
LIN {X -0.149,Y -671.232,Z 670.429,A 0.000,B 0.000,C 90.000,E1 293.206} C_DIS
LIN {X 0.221,Y -662.472,Z 670.428,A 0.000,B 0.000,C 90.000,E1 293.078} C_DIS
LIN {X -0.255,Y -655.535,Z 670.428,A 0.000,B 0.000,C 90.000,E1 293.025} C_DIS
LIN {X 0.029,Y -642.276,Z 670.427,A 0.000,B 0.000,C 90.000,E1 292.770} C_DIS
LIN {X -0.251,Y -632.403,Z 670.425,A 0.000,B 0.000,C 90.000,E1 292.589} C_DIS
LIN {X 0.354,Y -619.043,Z 670.424,A 0.000,B 0.000,C 90.000,E1 292.206} C_DIS
LIN {X -0.185,Y -601.991,Z 670.421,A 0.000,B 0.000,C 90.000,E1 291.770} C_DIS
LIN {X -0.029,Y -581.184,Z 670.417,A 0.000,B 0.000,C 90.000,E1 291.099} C_DIS
LIN {X 0.128,Y -575.716,Z 670.416,A 0.000,B 0.000,C 90.000,E1 290.918} C_DIS
LIN {X 0.188,Y -566.860,Z 670.415,A 0.000,B 0.000,C 90.000,E1 290.663} C_DIS
LIN {X -0.260,Y -563.568,Z 670.414,A 0.000,B 0.000,C 90.000,E1 290.610} C_DIS
LIN {X -0.053,Y -561.034,Z 670.414,A 0.000,B 0.000,C 90.000,E1 290.482} C_DIS
LIN {X 0.162,Y -556.529,Z 670.413,A 0.000,B 0.000,C 90.000,E1 290.248} C_DIS
LIN {X 0.114,Y -556.481,Z 670.413,A 0.000,B 0.000,C 90.000,E1 290.248} C_DIS
LIN {X -0.199,Y -555.307,Z 670.412,A 0.000,B 0.000,C 90.000,E1 290.120} C_DIS
LIN {X -0.241,Y -555.296,Z 670.412,A 0.000,B 0.000,C 90.000,E1 290.120} C_DIS
LIN {X 0.191,Y -554.645,Z 670.410,A 0.000,B 0.000,C 90.000,E1 289.758} C_DIS
LIN {X 0.216,Y -554.297,Z 670.404,A 0.000,B 0.000,C 90.000,E1 288.779} C_DIS
LIN {X 0.041,Y -554.022,Z 670.397,A 0.000,B 0.000,C 90.000,E1 287.402} C_DIS
LIN {X -0.134,Y -553.557,Z 670.389,A 0.000,B 0.000,C 90.000,E1 286.024} C_DIS
LIN {X -0.050,Y -553.164,Z 670.383,A 0.000,B 0.000,C 90.000,E1 284.898} C_DIS
LIN {X 0.028,Y -552.730,Z 670.377,A 0.000,B 0.000,C 90.000,E1 283.772} C_DIS
LIN {X -0.211,Y -551.792,Z 670.367,A 0.000,B 0.000,C 90.000,E1 282.119} C_DIS
LIN {X -0.043,Y -550.868,Z 670.356,A 0.000,B 0.000,C 90.000,E1 280.141} C_DIS
LIN {X -0.197,Y -549.940,Z 670.341,A 0.000,B 0.000,C 90.000,E1 277.352} C_DIS
LIN {X 0.176,Y -549.679,Z 670.333,A 0.000,B 0.000,C 90.000,E1 275.910} C_DIS
LIN {X 0.123,Y -549.435,Z 670.320,A 0.000,B 0.000,C 90.000,E1 273.669} C_DIS
LIN {X -0.144,Y -549.198,Z 670.313,A 0.000,B 0.000,C 90.000,E1 272.293} C_DIS
LIN {X 0.028,Y -548.948,Z 670.308,A 0.000,B 0.000,C 90.000,E1 271.432} C_DIS
LIN {X -0.264,Y -548.315,Z 670.300,A 0.000,B 0.000,C 90.000,E1 270.057} C_DIS
LIN {X -0.019,Y -547.555,Z 670.292,A 0.000,B 0.000,C 90.000,E1 268.625} C_DIS
LIN {X -0.285,Y -546.530,Z 670.283,A 0.000,B 0.000,C 90.000,E1 266.963} C_DIS
LIN {X -0.033,Y -545.623,Z 670.275,A 0.000,B 0.000,C 90.000,E1 265.527} C_DIS
LIN {X 0.205,Y -544.479,Z 670.267,A 0.000,B 0.000,C 90.000,E1 264.090} C_DIS
LIN {X -0.066,Y -543.206,Z 670.259,A 0.000,B 0.000,C 90.000,E1 262.704} C_DIS
LIN {X -0.286,Y -541.335,Z 670.250,A 0.000,B 0.000,C 90.000,E1 261.027} C_DIS
LIN {X -0.247,Y -538.928,Z 670.236,A 0.000,B 0.000,C 90.000,E1 258.465} C_DIS
LIN {X -0.127,Y -537.082,Z 670.223,A 0.000,B 0.000,C 90.000,E1 256.172} C_DIS
LIN {X -0.228,Y -535.808,Z 670.215,A 0.000,B 0.000,C 90.000,E1 254.755} C_DIS
LIN {X 0.256,Y -534.698,Z 670.209,A 0.000,B 0.000,C 90.000,E1 253.559} C_DIS
LIN {X 0.160,Y -532.397,Z 670.196,A 0.000,B 0.000,C 90.000,E1 251.275} C_DIS
LIN {X 0.078,Y -531.237,Z 670.190,A 0.000,B 0.000,C 90.000,E1 250.134} C_DIS
LIN {X 0.152,Y -530.143,Z 670.185,A 0.000,B 0.000,C 90.000,E1 249.263} C_DIS
LIN {X 0.089,Y -527.727,Z 670.175,A 0.000,B 0.000,C 90.000,E1 247.539} C_DIS
LIN {X -0.171,Y -526.080,Z 670.169,A 0.000,B 0.000,C 90.000,E1 246.410} C_DIS
LIN {X -0.129,Y -523.068,Z 670.159,A 0.000,B 0.000,C 90.000,E1 244.665} C_DIS
LIN {X -0.235,Y -520.928,Z 670.153,A 0.000,B 0.000,C 90.000,E1 243.512} C_DIS
LIN {X 0.126,Y -517.464,Z 670.143,A 0.000,B 0.000,C 90.000,E1 241.719} C_DIS
LIN {X 0.175,Y -515.042,Z 670.136,A 0.000,B 0.000,C 90.000,E1 240.539} C_DIS
LIN {X 0.094,Y -511.803,Z 670.128,A 0.000,B 0.000,C 90.000,E1 239.076} C_DIS
LIN {X 0.222,Y -508.577,Z 670.120,A 0.000,B 0.000,C 90.000,E1 237.582} C_DIS
LIN {X 0.184,Y -504.498,Z 670.110,A 0.000,B 0.000,C 90.000,E1 235.801} C_DIS
LIN {X 0.157,Y -501.538,Z 670.104,A 0.000,B 0.000,C 90.000,E1 234.609} C_DIS
LIN {X -0.167,Y -497.017,Z 670.094,A 0.000,B 0.000,C 90.000,E1 232.844} C_DIS
LIN {X -0.135,Y -491.889,Z 670.082,A 0.000,B 0.000,C 90.000,E1 230.723} C_DIS
LIN {X 0.247,Y -488.974,Z 670.075,A 0.000,B 0.000,C 90.000,E1 229.461} C_DIS
LIN {X 0.033,Y -485.328,Z 670.067,A 0.000,B 0.000,C 90.000,E1 227.957} C_DIS
LIN {X -0.021,Y -480.281,Z 670.055,A 0.000,B 0.000,C 90.000,E1 225.810} C_DIS
LIN {X 0.022,Y -475.838,Z 670.044,A 0.000,B 0.000,C 90.000,E1 223.947} C_DIS
LIN {X -0.020,Y -471.527,Z 670.034,A 0.000,B 0.000,C 90.000,E1 222.081} C_DIS
LIN {X 0.020,Y -466.151,Z 670.020,A 0.000,B 0.000,C 90.000,E1 219.564} C_DIS
LIN {X 0.121,Y -462.895,Z 670.011,A 0.000,B 0.000,C 90.000,E1 217.971} C_DIS
LIN {X 0.022,Y -457.767,Z 669.997,A 0.000,B 0.000,C 90.000,E1 215.438} C_DIS
LIN {X 0.157,Y -454.141,Z 669.986,A 0.000,B 0.000,C 90.000,E1 213.499} C_DIS
LIN {X -0.131,Y -451.101,Z 669.977,A 0.000,B 0.000,C 90.000,E1 211.926} C_DIS
LIN {X -0.176,Y -446.857,Z 669.965,A 0.000,B 0.000,C 90.000,E1 209.667} C_DIS
LIN {X -0.162,Y -442.808,Z 669.952,A 0.000,B 0.000,C 90.000,E1 207.385} C_DIS
LIN {X 0.053,Y -439.844,Z 669.943,A 0.000,B 0.000,C 90.000,E1 205.720} C_DIS
LIN {X 0.262,Y -435.763,Z 669.930,A 0.000,B 0.000,C 90.000,E1 203.387} C_DIS
LIN {X 0.194,Y -432.108,Z 669.919,A 0.000,B 0.000,C 90.000,E1 201.408} C_DIS
LIN {X -0.114,Y -428.514,Z 669.908,A 0.000,B 0.000,C 90.000,E1 199.450} C_DIS
LIN {X 0.141,Y -423.917,Z 669.893,A 0.000,B 0.000,C 90.000,E1 196.732} C_DIS
LIN {X 0.064,Y -420.518,Z 669.882,A 0.000,B 0.000,C 90.000,E1 194.717} C_DIS
LIN {X 0.107,Y -418.206,Z 669.874,A 0.000,B 0.000,C 90.000,E1 193.355} C_DIS
LIN {X -0.115,Y -413.776,Z 669.859,A 0.000,B 0.000,C 90.000,E1 190.658} C_DIS
LIN {X 0.086,Y -411.163,Z 669.850,A 0.000,B 0.000,C 90.000,E1 188.916} C_DIS
LIN {X 0.196,Y -408.041,Z 669.838,A 0.000,B 0.000,C 90.000,E1 186.834} C_DIS
LIN {X 0.105,Y -403.788,Z 669.821,A 0.000,B 0.000,C 90.000,E1 183.726} C_DIS
LIN {X -0.163,Y -400.486,Z 669.805,A 0.000,B 0.000,C 90.000,E1 180.974} C_DIS
LIN {X -0.138,Y -397.840,Z 669.790,A 0.000,B 0.000,C 90.000,E1 178.165} C_DIS
LIN {X 0.174,Y -395.592,Z 669.772,A 0.000,B 0.000,C 90.000,E1 174.951} C_DIS
LIN {X 0.106,Y -394.092,Z 669.754,A 0.000,B 0.000,C 90.000,E1 171.781} C_DIS
LIN {X -0.045,Y -393.628,Z 669.747,A 0.000,B 0.000,C 90.000,E1 170.387} C_DIS
LIN {X 0.176,Y -393.205,Z 669.735,A 0.000,B 0.000,C 90.000,E1 168.229} C_DIS
LIN {X 0.081,Y -393.026,Z 669.723,A 0.000,B 0.000,C 90.000,E1 166.117} C_DIS
LIN {X -0.211,Y -392.977,Z 669.707,A 0.000,B 0.000,C 90.000,E1 163.323} C_DIS
LIN {X 0.223,Y -393.202,Z 669.691,A 0.000,B 0.000,C 90.000,E1 160.423} C_DIS
LIN {X 0.015,Y -393.319,Z 669.686,A 0.000,B 0.000,C 90.000,E1 159.390} C_DIS
LIN {X -0.065,Y -393.641,Z 669.672,A 0.000,B 0.000,C 90.000,E1 156.922} C_DIS
LIN {X 0.172,Y -394.020,Z 669.658,A 0.000,B 0.000,C 90.000,E1 154.409} C_DIS
LIN {X -0.012,Y -394.378,Z 669.648,A 0.000,B 0.000,C 90.000,E1 152.666} C_DIS
LIN {X -0.187,Y -394.795,Z 669.638,A 0.000,B 0.000,C 90.000,E1 150.923} C_DIS
LIN {X -0.104,Y -395.286,Z 669.627,A 0.000,B 0.000,C 90.000,E1 148.791} C_DIS
LIN {X 0.202,Y -396.001,Z 669.615,A 0.000,B 0.000,C 90.000,E1 146.628} C_DIS
LIN {X 0.050,Y -397.297,Z 669.599,A 0.000,B 0.000,C 90.000,E1 143.829} C_DIS
LIN {X 0.096,Y -398.865,Z 669.583,A 0.000,B 0.000,C 90.000,E1 141.009} C_DIS
LIN {X 0.006,Y -400.497,Z 669.570,A 0.000,B 0.000,C 90.000,E1 138.566} C_DIS
LIN {X 0.131,Y -401.463,Z 669.562,A 0.000,B 0.000,C 90.000,E1 137.148} C_DIS
LIN {X -0.073,Y -402.961,Z 669.550,A 0.000,B 0.000,C 90.000,E1 135.081} C_DIS
LIN {X -0.021,Y -403.915,Z 669.545,A 0.000,B 0.000,C 90.000,E1 134.028} C_DIS
LIN {X -0.070,Y -404.699,Z 669.541,A 0.000,B 0.000,C 90.000,E1 133.338} C_DIS
LIN {X 0.166,Y -405.860,Z 669.537,A 0.000,B 0.000,C 90.000,E1 132.609} C_DIS
LIN {X -0.061,Y -407.550,Z 669.534,A 0.000,B 0.000,C 90.000,E1 132.043} C_DIS
LIN {X 0.009,Y -410.096,Z 669.531,A 0.000,B 0.000,C 90.000,E1 131.515} C_DIS
LIN {X 0.162,Y -412.679,Z 669.529,A 0.000,B 0.000,C 90.000,E1 131.148} C_DIS
LIN {X 0.110,Y -414.041,Z 669.528,A 0.000,B 0.000,C 90.000,E1 130.987} C_DIS
LIN {X 0.018,Y -418.915,Z 669.525,A 0.000,B 0.000,C 90.000,E1 130.539} C_DIS
LIN {X 0.077,Y -443.849,Z 669.514,A 0.000,B 0.000,C 90.000,E1 128.543} C_DIS
LIN {X 0.006,Y -456.496,Z 669.509,A 0.000,B 0.000,C 90.000,E1 127.604} C_DIS
LIN {X 0.135,Y -464.281,Z 669.506,A 0.000,B 0.000,C 90.000,E1 126.996} C_DIS
LIN {X 0.226,Y -470.476,Z 669.503,A 0.000,B 0.000,C 90.000,E1 126.503} C_DIS
LIN {X 0.072,Y -481.071,Z 669.498,A 0.000,B 0.000,C 90.000,E1 125.644} C_DIS
LIN {X 0.110,Y -488.102,Z 669.495,A 0.000,B 0.000,C 90.000,E1 125.025} C_DIS
LIN {X -0.015,Y -495.099,Z 669.491,A 0.000,B 0.000,C 90.000,E1 124.405} C_DIS
LIN {X 0.251,Y -502.169,Z 669.487,A 0.000,B 0.000,C 90.000,E1 123.706} C_DIS
LIN {X 0.180,Y -509.058,Z 669.484,A 0.000,B 0.000,C 90.000,E1 123.038} C_DIS
LIN {X 0.250,Y -515.795,Z 669.480,A 0.000,B 0.000,C 90.000,E1 122.339} C_DIS
LIN {X -0.123,Y -523.373,Z 669.475,A 0.000,B 0.000,C 90.000,E1 121.544} C_DIS
LIN {X 0.027,Y -528.963,Z 669.472,A 0.000,B 0.000,C 90.000,E1 120.875} C_DIS
LIN {X -0.289,Y -534.337,Z 669.468,A 0.000,B 0.000,C 90.000,E1 120.207} C_DIS
LIN {X -0.131,Y -538.332,Z 669.465,A 0.000,B 0.000,C 90.000,E1 119.617} C_DIS
LIN {X 0.185,Y -542.720,Z 669.461,A 0.000,B 0.000,C 90.000,E1 118.871} C_DIS
LIN {X 0.021,Y -546.656,Z 669.457,A 0.000,B 0.000,C 90.000,E1 118.180} C_DIS
LIN {X 0.153,Y -550.247,Z 669.453,A 0.000,B 0.000,C 90.000,E1 117.462} C_DIS
LIN {X -0.022,Y -555.323,Z 669.446,A 0.000,B 0.000,C 90.000,E1 116.360} C_DIS
LIN {X -0.169,Y -558.850,Z 669.442,A 0.000,B 0.000,C 90.000,E1 115.540} C_DIS
LIN {X 0.157,Y -561.043,Z 669.439,A 0.000,B 0.000,C 90.000,E1 114.951} C_DIS
LIN {X -0.135,Y -565.065,Z 669.433,A 0.000,B 0.000,C 90.000,E1 113.875} C_DIS
LIN {X -0.080,Y -568.532,Z 669.427,A 0.000,B 0.000,C 90.000,E1 112.770} C_DIS
LIN {X -0.103,Y -570.894,Z 669.422,A 0.000,B 0.000,C 90.000,E1 111.950} C_DIS
LIN {X 0.040,Y -573.581,Z 669.416,A 0.000,B 0.000,C 90.000,E1 110.844} C_DIS
LIN {X -0.150,Y -576.518,Z 669.408,A 0.000,B 0.000,C 90.000,E1 109.504} C_DIS
LIN {X 0.074,Y -579.251,Z 669.401,A 0.000,B 0.000,C 90.000,E1 108.127} C_DIS
LIN {X 0.190,Y -582.515,Z 669.392,A 0.000,B 0.000,C 90.000,E1 106.496} C_DIS
LIN {X -0.194,Y -585.156,Z 669.384,A 0.000,B 0.000,C 90.000,E1 105.190} C_DIS
LIN {X 0.033,Y -587.707,Z 669.377,A 0.000,B 0.000,C 90.000,E1 103.828} C_DIS
LIN {X 0.171,Y -590.251,Z 669.369,A 0.000,B 0.000,C 90.000,E1 102.479} C_DIS
LIN {X 0.048,Y -593.168,Z 669.361,A 0.000,B 0.000,C 90.000,E1 100.894} C_DIS
LIN {X 0.166,Y -595.651,Z 669.353,A 0.000,B 0.000,C 90.000,E1 99.557} C_DIS
LIN {X -0.063,Y -598.409,Z 669.344,A 0.000,B 0.000,C 90.000,E1 97.992} C_DIS
LIN {X 0.058,Y -600.413,Z 669.337,A 0.000,B 0.000,C 90.000,E1 96.663} C_DIS
LIN {X -0.088,Y -601.982,Z 669.331,A 0.000,B 0.000,C 90.000,E1 95.625} C_DIS
LIN {X -0.218,Y -603.494,Z 669.325,A 0.000,B 0.000,C 90.000,E1 94.588} C_DIS
LIN {X -0.122,Y -605.138,Z 669.318,A 0.000,B 0.000,C 90.000,E1 93.269} C_DIS
LIN {X -0.254,Y -606.297,Z 669.312,A 0.000,B 0.000,C 90.000,E1 92.236} C_DIS
LIN {X 0.227,Y -607.302,Z 669.307,A 0.000,B 0.000,C 90.000,E1 91.146} C_DIS
LIN {X -0.172,Y -607.871,Z 669.302,A 0.000,B 0.000,C 90.000,E1 90.401} C_DIS
LIN {X -0.290,Y -608.534,Z 669.296,A 0.000,B 0.000,C 90.000,E1 89.370} C_DIS
LIN {X 0.206,Y -608.898,Z 669.291,A 0.000,B 0.000,C 90.000,E1 88.282} C_DIS
LIN {X 0.114,Y -609.245,Z 669.285,A 0.000,B 0.000,C 90.000,E1 87.249} C_DIS
LIN {X -0.305,Y -609.404,Z 669.278,A 0.000,B 0.000,C 90.000,E1 85.988} C_DIS
LIN {X -0.005,Y -609.305,Z 669.273,A 0.000,B 0.000,C 90.000,E1 85.179} C_DIS
LIN {X 0.233,Y -609.067,Z 669.266,A 0.000,B 0.000,C 90.000,E1 83.856} C_DIS
LIN {X -0.150,Y -608.535,Z 669.259,A 0.000,B 0.000,C 90.000,E1 82.591} C_DIS
LIN {X 0.157,Y -608.159,Z 669.254,A 0.000,B 0.000,C 90.000,E1 81.781} C_DIS
LIN {X 0.189,Y -607.405,Z 669.249,A 0.000,B 0.000,C 90.000,E1 80.735} C_DIS
LIN {X -0.055,Y -606.066,Z 669.241,A 0.000,B 0.000,C 90.000,E1 79.454} C_DIS
LIN {X 0.334,Y -605.189,Z 669.237,A 0.000,B 0.000,C 90.000,E1 78.634} C_DIS
LIN {X -0.272,Y -603.952,Z 669.231,A 0.000,B 0.000,C 90.000,E1 77.645} C_DIS
LIN {X -0.181,Y -602.557,Z 669.225,A 0.000,B 0.000,C 90.000,E1 76.589} C_DIS
LIN {X 0.033,Y -601.067,Z 669.220,A 0.000,B 0.000,C 90.000,E1 75.519} C_DIS
LIN {X 0.234,Y -599.514,Z 669.214,A 0.000,B 0.000,C 90.000,E1 74.448} C_DIS
LIN {X 0.122,Y -597.357,Z 669.206,A 0.000,B 0.000,C 90.000,E1 73.142} C_DIS
LIN {X -0.011,Y -595.974,Z 669.202,A 0.000,B 0.000,C 90.000,E1 72.362} C_DIS
LIN {X 0.288,Y -594.074,Z 669.196,A 0.000,B 0.000,C 90.000,E1 71.275} C_DIS
LIN {X -0.316,Y -591.444,Z 669.189,A 0.000,B 0.000,C 90.000,E1 70.007} C_DIS
LIN {X -0.318,Y -589.710,Z 669.184,A 0.000,B 0.000,C 90.000,E1 69.209} C_DIS
LIN {X 0.091,Y -587.119,Z 669.178,A 0.000,B 0.000,C 90.000,E1 68.103} C_DIS
LIN {X -0.151,Y -585.715,Z 669.175,A 0.000,B 0.000,C 90.000,E1 67.592} C_DIS
LIN {X -0.211,Y -583.337,Z 669.171,A 0.000,B 0.000,C 90.000,E1 66.794} C_DIS
LIN {X 0.066,Y -581.755,Z 669.168,A 0.000,B 0.000,C 90.000,E1 66.230} C_DIS
LIN {X 0.194,Y -579.106,Z 669.164,A 0.000,B 0.000,C 90.000,E1 65.409} C_DIS
LIN {X 0.293,Y -576.290,Z 669.159,A 0.000,B 0.000,C 90.000,E1 64.588} C_DIS
LIN {X 0.202,Y -572.196,Z 669.153,A 0.000,B 0.000,C 90.000,E1 63.512} C_DIS
LIN {X -0.287,Y -568.946,Z 669.148,A 0.000,B 0.000,C 90.000,E1 62.743} C_DIS
LIN {X -0.041,Y -565.388,Z 669.144,A 0.000,B 0.000,C 90.000,E1 61.897} C_DIS
LIN {X 0.256,Y -562.217,Z 669.140,A 0.000,B 0.000,C 90.000,E1 61.179} C_DIS
LIN {X -0.140,Y -559.484,Z 669.137,A 0.000,B 0.000,C 90.000,E1 60.667} C_DIS
LIN {X 0.097,Y -555.519,Z 669.133,A 0.000,B 0.000,C 90.000,E1 59.950} C_DIS
LIN {X -0.174,Y -551.062,Z 669.129,A 0.000,B 0.000,C 90.000,E1 59.282} C_DIS
LIN {X 0.273,Y -546.063,Z 669.125,A 0.000,B 0.000,C 90.000,E1 58.535} C_DIS
LIN {X 0.261,Y -543.006,Z 669.123,A 0.000,B 0.000,C 90.000,E1 58.122} C_DIS
LIN {X 0.239,Y -538.505,Z 669.120,A 0.000,B 0.000,C 90.000,E1 57.582} C_DIS
LIN {X 0.207,Y -533.407,Z 669.117,A 0.000,B 0.000,C 90.000,E1 57.041} C_DIS
LIN {X -0.341,Y -529.162,Z 669.115,A 0.000,B 0.000,C 90.000,E1 56.707} C_DIS
LIN {X -0.116,Y -523.690,Z 669.112,A 0.000,B 0.000,C 90.000,E1 56.215} C_DIS
LIN {X 0.119,Y -517.417,Z 669.110,A 0.000,B 0.000,C 90.000,E1 55.722} C_DIS
LIN {X 0.092,Y -512.382,Z 669.108,A 0.000,B 0.000,C 90.000,E1 55.388} C_DIS
LIN {X 0.076,Y -504.217,Z 669.105,A 0.000,B 0.000,C 90.000,E1 54.895} C_DIS
LIN {X 0.000,Y -497.672,Z 669.103,A 0.000,B 0.000,C 90.000,E1 54.529} C_DIS
LIN {X -0.045,Y -480.950,Z 669.098,A 0.000,B 0.000,C 90.000,E1 53.623} C_DIS
LIN {X -0.114,Y -464.347,Z 669.093,A 0.000,B 0.000,C 90.000,E1 52.718} C_DIS
LIN {X 0.071,Y -441.533,Z 669.086,A 0.000,B 0.000,C 90.000,E1 51.376} C_DIS
LIN {X 0.232,Y -431.396,Z 669.082,A 0.000,B 0.000,C 90.000,E1 50.723} C_DIS
LIN {X 0.209,Y -431.363,Z 669.082,A 0.000,B 0.000,C 90.000,E1 50.723} C_DIS
LIN {X 0.085,Y -421.804,Z 669.059,A 0.000,B 0.000,C 90.000,E1 46.539} C_DIS
LIN {X 0.149,Y -418.707,Z 669.049,A 0.000,B 0.000,C 90.000,E1 44.838} C_DIS
LIN {X -0.108,Y -416.894,Z 669.045,A 0.000,B 0.000,C 90.000,E1 44.109} C_DIS
LIN {X 0.079,Y -416.961,Z 669.034,A 0.000,B 0.000,C 90.000,E1 42.123} C_DIS
LIN {X 0.042,Y -417.361,Z 669.019,A 0.000,B 0.000,C 90.000,E1 39.402} C_DIS
LIN {X -0.047,Y -418.697,Z 669.000,A 0.000,B 0.000,C 90.000,E1 36.011} C_DIS
LIN {X 0.047,Y -419.285,Z 668.994,A 0.000,B 0.000,C 90.000,E1 34.978} C_DIS
LIN {X -0.121,Y -420.430,Z 668.981,A 0.000,B 0.000,C 90.000,E1 32.625} C_DIS
LIN {X -0.108,Y -421.527,Z 668.970,A 0.000,B 0.000,C 90.000,E1 30.590} C_DIS
LIN {X 0.130,Y -422.261,Z 668.962,A 0.000,B 0.000,C 90.000,E1 29.205} C_DIS
LIN {X -0.105,Y -423.693,Z 668.949,A 0.000,B 0.000,C 90.000,E1 26.873} C_DIS
LIN {X -0.113,Y -425.267,Z 668.936,A 0.000,B 0.000,C 90.000,E1 24.515} C_DIS
LIN {X -0.237,Y -427.714,Z 668.921,A 0.000,B 0.000,C 90.000,E1 21.844} C_DIS
LIN {X 0.133,Y -429.275,Z 668.912,A 0.000,B 0.000,C 90.000,E1 20.120} C_DIS
LIN {X -0.046,Y -430.108,Z 668.906,A 0.000,B 0.000,C 90.000,E1 19.141} C_DIS
LIN {X 0.080,Y -431.285,Z 668.897,A 0.000,B 0.000,C 90.000,E1 17.457} C_DIS
LIN {X -0.089,Y -432.755,Z 668.886,A 0.000,B 0.000,C 90.000,E1 15.481} C_DIS
LIN {X -0.027,Y -434.538,Z 668.875,A 0.000,B 0.000,C 90.000,E1 13.480} C_DIS
LIN {X 0.083,Y -436.518,Z 668.864,A 0.000,B 0.000,C 90.000,E1 11.478} C_DIS
LIN {X 0.072,Y -439.669,Z 668.847,A 0.000,B 0.000,C 90.000,E1 8.511} C_DIS
LIN {X -0.127,Y -442.806,Z 668.833,A 0.000,B 0.000,C 90.000,E1 5.910} C_DIS
LIN {X -0.057,Y -447.210,Z 668.815,A 0.000,B 0.000,C 90.000,E1 2.636} C_DIS
LIN {X 0.107,Y -450.524,Z 668.802,A 0.000,B 0.000,C 90.000,E1 0.344} C_DIS
LIN {X 0.112,Y -454.174,Z 668.790,A 0.000,B 0.000,C 90.000,E1 358.165} C_DIS
LIN {X 0.047,Y -458.175,Z 668.777,A 0.000,B 0.000,C 90.000,E1 355.927} C_DIS
LIN {X -0.126,Y -461.704,Z 668.767,A 0.000,B 0.000,C 90.000,E1 354.033} C_DIS
LIN {X -0.135,Y -465.216,Z 668.756,A 0.000,B 0.000,C 90.000,E1 352.129} C_DIS
LIN {X -0.003,Y -467.544,Z 668.749,A 0.000,B 0.000,C 90.000,E1 350.849} C_DIS
LIN {X -0.094,Y -470.394,Z 668.740,A 0.000,B 0.000,C 90.000,E1 349.285} C_DIS
LIN {X 0.162,Y -474.270,Z 668.728,A 0.000,B 0.000,C 90.000,E1 347.061} C_DIS
LIN {X 0.026,Y -477.126,Z 668.720,A 0.000,B 0.000,C 90.000,E1 345.519} C_DIS
LIN {X -0.205,Y -480.625,Z 668.709,A 0.000,B 0.000,C 90.000,E1 343.685} C_DIS
LIN {X -0.088,Y -484.809,Z 668.697,A 0.000,B 0.000,C 90.000,E1 341.511} C_DIS
LIN {X 0.122,Y -488.508,Z 668.687,A 0.000,B 0.000,C 90.000,E1 339.645} C_DIS
LIN {X -0.164,Y -492.214,Z 668.677,A 0.000,B 0.000,C 90.000,E1 337.847} C_DIS
LIN {X 0.041,Y -495.088,Z 668.668,A 0.000,B 0.000,C 90.000,E1 336.305} C_DIS
LIN {X -0.011,Y -497.279,Z 668.662,A 0.000,B 0.000,C 90.000,E1 335.101} C_DIS
LIN {X -0.078,Y -501.259,Z 668.650,A 0.000,B 0.000,C 90.000,E1 332.999} C_DIS
LIN {X -0.109,Y -503.430,Z 668.645,A 0.000,B 0.000,C 90.000,E1 332.103} C_DIS
LIN {X 0.192,Y -504.423,Z 668.643,A 0.000,B 0.000,C 90.000,E1 331.769} C_DIS
LIN {X 0.126,Y -507.146,Z 668.640,A 0.000,B 0.000,C 90.000,E1 331.179} C_DIS
LIN {X 0.059,Y -510.292,Z 668.637,A 0.000,B 0.000,C 90.000,E1 330.717} C_DIS
LIN {X -0.114,Y -512.254,Z 668.636,A 0.000,B 0.000,C 90.000,E1 330.511} C_DIS
LIN {X 0.010,Y -519.475,Z 668.633,A 0.000,B 0.000,C 90.000,E1 329.871} C_DIS
LIN {X -0.244,Y -531.123,Z 668.628,A 0.000,B 0.000,C 90.000,E1 329.076} C_DIS
LIN {X -0.126,Y -541.656,Z 668.624,A 0.000,B 0.000,C 90.000,E1 328.280} C_DIS
LIN {X 0.152,Y -547.341,Z 668.621,A 0.000,B 0.000,C 90.000,E1 327.788} C_DIS
LIN {X -0.068,Y -557.140,Z 668.616,A 0.000,B 0.000,C 90.000,E1 326.962} C_DIS
LIN {X 0.367,Y -562.527,Z 668.614,A 0.000,B 0.000,C 90.000,E1 326.421} C_DIS
LIN {X -0.024,Y -573.062,Z 668.608,A 0.000,B 0.000,C 90.000,E1 325.435} C_DIS
LIN {X 0.148,Y -583.369,Z 668.602,A 0.000,B 0.000,C 90.000,E1 324.402} C_DIS
LIN {X 0.197,Y -592.244,Z 668.597,A 0.000,B 0.000,C 90.000,E1 323.497} C_DIS
LIN {X 0.178,Y -599.641,Z 668.593,A 0.000,B 0.000,C 90.000,E1 322.718} C_DIS
LIN {X 0.156,Y -605.549,Z 668.589,A 0.000,B 0.000,C 90.000,E1 322.065} C_DIS
LIN {X 0.210,Y -610.088,Z 668.586,A 0.000,B 0.000,C 90.000,E1 321.537} C_DIS
LIN {X -0.271,Y -616.325,Z 668.582,A 0.000,B 0.000,C 90.000,E1 320.803} C_DIS
LIN {X -0.181,Y -621.208,Z 668.579,A 0.000,B 0.000,C 90.000,E1 320.150} C_DIS
LIN {X -0.016,Y -624.892,Z 668.576,A 0.000,B 0.000,C 90.000,E1 319.622} C_DIS
LIN {X 0.086,Y -630.917,Z 668.571,A 0.000,B 0.000,C 90.000,E1 318.728} C_DIS
LIN {X 0.240,Y -634.999,Z 668.567,A 0.000,B 0.000,C 90.000,E1 318.081} C_DIS
LIN {X -0.089,Y -640.509,Z 668.562,A 0.000,B 0.000,C 90.000,E1 317.229} C_DIS
LIN {X 0.061,Y -646.437,Z 668.557,A 0.000,B 0.000,C 90.000,E1 316.215} C_DIS
LIN {X -0.179,Y -652.046,Z 668.551,A 0.000,B 0.000,C 90.000,E1 315.243} C_DIS
LIN {X 0.171,Y -655.401,Z 668.548,A 0.000,B 0.000,C 90.000,E1 314.595} C_DIS
LIN {X 0.101,Y -658.008,Z 668.545,A 0.000,B 0.000,C 90.000,E1 314.109} C_DIS
LIN {X -0.014,Y -664.032,Z 668.538,A 0.000,B 0.000,C 90.000,E1 312.894} C_DIS
LIN {X -0.023,Y -666.927,Z 668.535,A 0.000,B 0.000,C 90.000,E1 312.285} C_DIS
LIN {X 0.027,Y -671.402,Z 668.530,A 0.000,B 0.000,C 90.000,E1 311.310} C_DIS
LIN {X -0.386,Y -674.571,Z 668.526,A 0.000,B 0.000,C 90.000,E1 310.620} C_DIS
LIN {X -0.233,Y -678.457,Z 668.520,A 0.000,B 0.000,C 90.000,E1 309.644} C_DIS
LIN {X 0.340,Y -680.256,Z 668.518,A 0.000,B 0.000,C 90.000,E1 309.116} C_DIS
LIN {X 0.171,Y -684.185,Z 668.511,A 0.000,B 0.000,C 90.000,E1 307.935} C_DIS
LIN {X -0.021,Y -686.351,Z 668.507,A 0.000,B 0.000,C 90.000,E1 307.237} C_DIS
LIN {X 0.447,Y -689.499,Z 668.500,A 0.000,B 0.000,C 90.000,E1 306.011} C_DIS
LIN {X -0.046,Y -691.854,Z 668.495,A 0.000,B 0.000,C 90.000,E1 305.105} C_DIS
LIN {X 0.454,Y -693.930,Z 668.490,A 0.000,B 0.000,C 90.000,E1 304.119} C_DIS
LIN {X 0.010,Y -695.838,Z 668.485,A 0.000,B 0.000,C 90.000,E1 303.214} C_DIS
LIN {X 0.168,Y -697.546,Z 668.479,A 0.000,B 0.000,C 90.000,E1 302.260} C_DIS
LIN {X -0.360,Y -699.348,Z 668.473,A 0.000,B 0.000,C 90.000,E1 301.131} C_DIS
LIN {X 0.176,Y -700.350,Z 668.469,A 0.000,B 0.000,C 90.000,E1 300.384} C_DIS
LIN {X 0.028,Y -701.378,Z 668.464,A 0.000,B 0.000,C 90.000,E1 299.461} C_DIS
LIN {X -0.109,Y -702.329,Z 668.459,A 0.000,B 0.000,C 90.000,E1 298.537} C_DIS
LIN {X -0.004,Y -703.589,Z 668.451,A 0.000,B 0.000,C 90.000,E1 297.129} C_DIS
LIN {X 0.192,Y -704.390,Z 668.446,A 0.000,B 0.000,C 90.000,E1 296.181} C_DIS
LIN {X 0.132,Y -704.665,Z 668.443,A 0.000,B 0.000,C 90.000,E1 295.720} C_DIS
LIN {X 0.419,Y -704.611,Z 668.442,A 0.000,B 0.000,C 90.000,E1 295.463} C_DIS
LIN {X 0.055,Y -704.088,Z 668.439,A 0.000,B 0.000,C 90.000,E1 295.027} C_DIS
LIN {X 0.341,Y -703.369,Z 668.438,A 0.000,B 0.000,C 90.000,E1 294.771} C_DIS
LIN {X -0.167,Y -701.680,Z 668.436,A 0.000,B 0.000,C 90.000,E1 294.463} C_DIS
LIN {X 0.111,Y -700.276,Z 668.435,A 0.000,B 0.000,C 90.000,E1 294.207} C_DIS
LIN {X 0.248,Y -699.124,Z 668.434,A 0.000,B 0.000,C 90.000,E1 294.079} C_DIS
LIN {X -0.024,Y -694.324,Z 668.432,A 0.000,B 0.000,C 90.000,E1 293.770} C_DIS
LIN {X 0.355,Y -692.746,Z 668.432,A 0.000,B 0.000,C 90.000,E1 293.643} C_DIS
LIN {X -0.106,Y -690.923,Z 668.431,A 0.000,B 0.000,C 90.000,E1 293.590} C_DIS
LIN {X -0.289,Y -687.970,Z 668.431,A 0.000,B 0.000,C 90.000,E1 293.515} C_DIS
LIN {X 0.124,Y -681.323,Z 668.430,A 0.000,B 0.000,C 90.000,E1 293.334} C_DIS
LIN {X -0.347,Y -679.092,Z 668.430,A 0.000,B 0.000,C 90.000,E1 293.334} C_DIS
LIN {X -0.110,Y -669.600,Z 668.429,A 0.000,B 0.000,C 90.000,E1 293.206} C_DIS
LIN {X 0.012,Y -659.362,Z 668.428,A 0.000,B 0.000,C 90.000,E1 293.078} C_DIS
LIN {X -0.278,Y -649.540,Z 668.427,A 0.000,B 0.000,C 90.000,E1 292.950} C_DIS
LIN {X 0.311,Y -636.137,Z 668.426,A 0.000,B 0.000,C 90.000,E1 292.642} C_DIS
LIN {X 0.273,Y -622.884,Z 668.424,A 0.000,B 0.000,C 90.000,E1 292.333} C_DIS
LIN {X -0.026,Y -606.197,Z 668.422,A 0.000,B 0.000,C 90.000,E1 291.897} C_DIS
LIN {X -0.162,Y -578.527,Z 668.417,A 0.000,B 0.000,C 90.000,E1 291.046} C_DIS
LIN {X 0.216,Y -564.493,Z 668.415,A 0.000,B 0.000,C 90.000,E1 290.610} C_DIS
LIN {X -0.100,Y -561.632,Z 668.414,A 0.000,B 0.000,C 90.000,E1 290.536} C_DIS
LIN {X -0.251,Y -556.380,Z 668.413,A 0.000,B 0.000,C 90.000,E1 290.301} C_DIS
LIN {X 0.222,Y -556.341,Z 668.413,A 0.000,B 0.000,C 90.000,E1 290.248} C_DIS
LIN {X -0.082,Y -555.235,Z 668.412,A 0.000,B 0.000,C 90.000,E1 290.120} C_DIS
LIN {X -0.197,Y -554.950,Z 668.411,A 0.000,B 0.000,C 90.000,E1 289.993} C_DIS
LIN {X 0.089,Y -554.640,Z 668.410,A 0.000,B 0.000,C 90.000,E1 289.704} C_DIS
LIN {X -0.286,Y -554.339,Z 668.405,A 0.000,B 0.000,C 90.000,E1 288.906} C_DIS
LIN {X -0.038,Y -554.176,Z 668.399,A 0.000,B 0.000,C 90.000,E1 287.764} C_DIS
LIN {X -0.208,Y -553.779,Z 668.391,A 0.000,B 0.000,C 90.000,E1 286.386} C_DIS
LIN {X 0.143,Y -553.258,Z 668.383,A 0.000,B 0.000,C 90.000,E1 284.954} C_DIS
LIN {X 0.221,Y -552.833,Z 668.377,A 0.000,B 0.000,C 90.000,E1 283.828} C_DIS
LIN {X 0.096,Y -551.756,Z 668.366,A 0.000,B 0.000,C 90.000,E1 281.883} C_DIS
LIN {X 0.260,Y -550.834,Z 668.355,A 0.000,B 0.000,C 90.000,E1 279.905} C_DIS
LIN {X -0.009,Y -550.029,Z 668.341,A 0.000,B 0.000,C 90.000,E1 277.409} C_DIS
LIN {X -0.183,Y -549.761,Z 668.333,A 0.000,B 0.000,C 90.000,E1 276.024} C_DIS
LIN {X -0.237,Y -549.508,Z 668.321,A 0.000,B 0.000,C 90.000,E1 273.784} C_DIS
LIN {X -0.007,Y -549.324,Z 668.315,A 0.000,B 0.000,C 90.000,E1 272.636} C_DIS
LIN {X 0.217,Y -549.010,Z 668.308,A 0.000,B 0.000,C 90.000,E1 271.489} C_DIS
LIN {X -0.075,Y -548.383,Z 668.301,A 0.000,B 0.000,C 90.000,E1 270.115} C_DIS
LIN {X 0.171,Y -547.628,Z 668.293,A 0.000,B 0.000,C 90.000,E1 268.682} C_DIS
LIN {X -0.177,Y -546.971,Z 668.287,A 0.000,B 0.000,C 90.000,E1 267.593} C_DIS
LIN {X 0.018,Y -546.290,Z 668.280,A 0.000,B 0.000,C 90.000,E1 266.445} C_DIS
LIN {X 0.195,Y -545.539,Z 668.274,A 0.000,B 0.000,C 90.000,E1 265.298} C_DIS
LIN {X -0.059,Y -544.362,Z 668.266,A 0.000,B 0.000,C 90.000,E1 263.913} C_DIS
LIN {X 0.136,Y -543.315,Z 668.260,A 0.000,B 0.000,C 90.000,E1 262.761} C_DIS
LIN {X -0.079,Y -541.485,Z 668.250,A 0.000,B 0.000,C 90.000,E1 261.084} C_DIS
LIN {X -0.033,Y -539.064,Z 668.236,A 0.000,B 0.000,C 90.000,E1 258.522} C_DIS
LIN {X 0.095,Y -537.183,Z 668.224,A 0.000,B 0.000,C 90.000,E1 256.228} C_DIS
LIN {X -0.001,Y -535.937,Z 668.216,A 0.000,B 0.000,C 90.000,E1 254.810} C_DIS
LIN {X -0.176,Y -534.842,Z 668.209,A 0.000,B 0.000,C 90.000,E1 253.685} C_DIS
LIN {X 0.011,Y -533.086,Z 668.200,A 0.000,B 0.000,C 90.000,E1 251.945} C_DIS
LIN {X 0.114,Y -532.007,Z 668.193,A 0.000,B 0.000,C 90.000,E1 250.786} C_DIS
LIN {X 0.025,Y -530.705,Z 668.187,A 0.000,B 0.000,C 90.000,E1 249.645} C_DIS
LIN {X -0.035,Y -528.296,Z 668.177,A 0.000,B 0.000,C 90.000,E1 247.922} C_DIS
LIN {X -0.117,Y -526.269,Z 668.169,A 0.000,B 0.000,C 90.000,E1 246.485} C_DIS
LIN {X 0.143,Y -523.248,Z 668.160,A 0.000,B 0.000,C 90.000,E1 244.717} C_DIS
LIN {X 0.133,Y -521.701,Z 668.155,A 0.000,B 0.000,C 90.000,E1 243.845} C_DIS
LIN {X -0.085,Y -518.805,Z 668.147,A 0.000,B 0.000,C 90.000,E1 242.410} C_DIS
LIN {X 0.109,Y -515.824,Z 668.139,A 0.000,B 0.000,C 90.000,E1 240.923} C_DIS
LIN {X 0.046,Y -512.641,Z 668.130,A 0.000,B 0.000,C 90.000,E1 239.459} C_DIS
LIN {X -0.073,Y -509.406,Z 668.122,A 0.000,B 0.000,C 90.000,E1 237.995} C_DIS
LIN {X -0.092,Y -505.352,Z 668.112,A 0.000,B 0.000,C 90.000,E1 236.215} C_DIS
LIN {X -0.104,Y -502.485,Z 668.106,A 0.000,B 0.000,C 90.000,E1 235.022} C_DIS
LIN {X -0.001,Y -497.935,Z 668.096,A 0.000,B 0.000,C 90.000,E1 233.210} C_DIS
LIN {X -0.098,Y -492.045,Z 668.082,A 0.000,B 0.000,C 90.000,E1 230.803} C_DIS
LIN {X -0.248,Y -488.396,Z 668.074,A 0.000,B 0.000,C 90.000,E1 229.299} C_DIS
LIN {X 0.073,Y -485.492,Z 668.067,A 0.000,B 0.000,C 90.000,E1 228.038} C_DIS
LIN {X 0.022,Y -480.428,Z 668.055,A 0.000,B 0.000,C 90.000,E1 225.891} C_DIS
LIN {X -0.045,Y -476.731,Z 668.046,A 0.000,B 0.000,C 90.000,E1 224.352} C_DIS
LIN {X 0.254,Y -472.373,Z 668.036,A 0.000,B 0.000,C 90.000,E1 222.447} C_DIS
LIN {X 0.074,Y -466.236,Z 668.020,A 0.000,B 0.000,C 90.000,E1 219.644} C_DIS
LIN {X -0.186,Y -463.000,Z 668.012,A 0.000,B 0.000,C 90.000,E1 218.096} C_DIS
LIN {X 0.087,Y -457.877,Z 667.997,A 0.000,B 0.000,C 90.000,E1 215.518} C_DIS
LIN {X -0.053,Y -453.621,Z 667.985,A 0.000,B 0.000,C 90.000,E1 213.293} C_DIS
LIN {X 0.121,Y -449.983,Z 667.974,A 0.000,B 0.000,C 90.000,E1 211.337} C_DIS
LIN {X 0.049,Y -445.793,Z 667.962,A 0.000,B 0.000,C 90.000,E1 209.077} C_DIS
LIN {X -0.019,Y -442.269,Z 667.951,A 0.000,B 0.000,C 90.000,E1 207.129} C_DIS
LIN {X 0.152,Y -439.950,Z 667.943,A 0.000,B 0.000,C 90.000,E1 205.796} C_DIS
LIN {X 0.139,Y -436.440,Z 667.932,A 0.000,B 0.000,C 90.000,E1 203.823} C_DIS
LIN {X 0.087,Y -432.828,Z 667.921,A 0.000,B 0.000,C 90.000,E1 201.844} C_DIS
LIN {X 0.015,Y -428.597,Z 667.909,A 0.000,B 0.000,C 90.000,E1 199.523} C_DIS
LIN {X -0.121,Y -424.032,Z 667.894,A 0.000,B 0.000,C 90.000,E1 196.858} C_DIS
LIN {X -0.079,Y -420.639,Z 667.882,A 0.000,B 0.000,C 90.000,E1 194.828} C_DIS
LIN {X -0.039,Y -418.346,Z 667.875,A 0.000,B 0.000,C 90.000,E1 193.467} C_DIS
LIN {X 0.144,Y -413.932,Z 667.860,A 0.000,B 0.000,C 90.000,E1 190.715} C_DIS
LIN {X -0.061,Y -411.323,Z 667.850,A 0.000,B 0.000,C 90.000,E1 189.029} C_DIS
LIN {X 0.028,Y -408.744,Z 667.841,A 0.000,B 0.000,C 90.000,E1 187.296} C_DIS
LIN {X -0.034,Y -404.367,Z 667.823,A 0.000,B 0.000,C 90.000,E1 184.188} C_DIS
LIN {X 0.181,Y -401.421,Z 667.810,A 0.000,B 0.000,C 90.000,E1 181.718} C_DIS
LIN {X 0.168,Y -398.270,Z 667.792,A 0.000,B 0.000,C 90.000,E1 178.568} C_DIS
LIN {X 0.086,Y -395.955,Z 667.775,A 0.000,B 0.000,C 90.000,E1 175.412} C_DIS
LIN {X 0.028,Y -394.383,Z 667.757,A 0.000,B 0.000,C 90.000,E1 172.243} C_DIS
LIN {X 0.160,Y -393.582,Z 667.743,A 0.000,B 0.000,C 90.000,E1 169.746} C_DIS
LIN {X -0.007,Y -393.272,Z 667.731,A 0.000,B 0.000,C 90.000,E1 167.645} C_DIS
LIN {X -0.055,Y -393.120,Z 667.722,A 0.000,B 0.000,C 90.000,E1 165.880} C_DIS
LIN {X 0.145,Y -393.119,Z 667.706,A 0.000,B 0.000,C 90.000,E1 163.015} C_DIS
LIN {X 0.034,Y -393.391,Z 667.692,A 0.000,B 0.000,C 90.000,E1 160.550} C_DIS
LIN {X -0.172,Y -393.523,Z 667.686,A 0.000,B 0.000,C 90.000,E1 159.518} C_DIS
LIN {X 0.113,Y -393.847,Z 667.672,A 0.000,B 0.000,C 90.000,E1 156.997} C_DIS
LIN {X -0.008,Y -394.246,Z 667.659,A 0.000,B 0.000,C 90.000,E1 154.537} C_DIS
LIN {X 0.163,Y -394.621,Z 667.649,A 0.000,B 0.000,C 90.000,E1 152.743} C_DIS
LIN {X -0.149,Y -395.086,Z 667.637,A 0.000,B 0.000,C 90.000,E1 150.667} C_DIS
LIN {X 0.071,Y -395.545,Z 667.627,A 0.000,B 0.000,C 90.000,E1 148.869} C_DIS
LIN {X -0.083,Y -396.347,Z 667.613,A 0.000,B 0.000,C 90.000,E1 146.421} C_DIS
LIN {X 0.095,Y -397.636,Z 667.598,A 0.000,B 0.000,C 90.000,E1 143.577} C_DIS
LIN {X -0.174,Y -399.206,Z 667.582,A 0.000,B 0.000,C 90.000,E1 140.803} C_DIS
LIN {X -0.111,Y -400.612,Z 667.570,A 0.000,B 0.000,C 90.000,E1 138.690} C_DIS
LIN {X -0.252,Y -401.512,Z 667.563,A 0.000,B 0.000,C 90.000,E1 137.310} C_DIS
LIN {X -0.061,Y -403.215,Z 667.549,A 0.000,B 0.000,C 90.000,E1 134.838} C_DIS
LIN {X -0.178,Y -404.492,Z 667.541,A 0.000,B 0.000,C 90.000,E1 133.461} C_DIS
LIN {X -0.222,Y -405.477,Z 667.537,A 0.000,B 0.000,C 90.000,E1 132.771} C_DIS
LIN {X 0.183,Y -406.253,Z 667.536,A 0.000,B 0.000,C 90.000,E1 132.366} C_DIS
LIN {X -0.032,Y -407.618,Z 667.533,A 0.000,B 0.000,C 90.000,E1 131.881} C_DIS
LIN {X 0.230,Y -407.790,Z 667.532,A 0.000,B 0.000,C 90.000,E1 131.757} C_DIS
LIN {X 0.069,Y -409.424,Z 667.530,A 0.000,B 0.000,C 90.000,E1 131.434} C_DIS
LIN {X -0.010,Y -410.412,Z 667.529,A 0.000,B 0.000,C 90.000,E1 131.272} C_DIS
LIN {X 0.087,Y -412.969,Z 667.527,A 0.000,B 0.000,C 90.000,E1 130.906} C_DIS
LIN {X 0.010,Y -418.082,Z 667.525,A 0.000,B 0.000,C 90.000,E1 130.415} C_DIS
LIN {X 0.017,Y -431.972,Z 667.518,A 0.000,B 0.000,C 90.000,E1 129.277} C_DIS
LIN {X -0.139,Y -452.754,Z 667.510,A 0.000,B 0.000,C 90.000,E1 127.729} C_DIS
LIN {X -0.255,Y -460.639,Z 667.506,A 0.000,B 0.000,C 90.000,E1 127.156} C_DIS
LIN {X -0.128,Y -469.997,Z 667.502,A 0.000,B 0.000,C 90.000,E1 126.423} C_DIS
LIN {X 0.222,Y -480.545,Z 667.497,A 0.000,B 0.000,C 90.000,E1 125.518} C_DIS
LIN {X 0.105,Y -487.877,Z 667.494,A 0.000,B 0.000,C 90.000,E1 124.898} C_DIS
LIN {X 0.003,Y -494.877,Z 667.490,A 0.000,B 0.000,C 90.000,E1 124.278} C_DIS
LIN {X -0.085,Y -501.970,Z 667.487,A 0.000,B 0.000,C 90.000,E1 123.627} C_DIS
LIN {X -0.163,Y -508.907,Z 667.483,A 0.000,B 0.000,C 90.000,E1 122.959} C_DIS
LIN {X -0.049,Y -515.621,Z 667.479,A 0.000,B 0.000,C 90.000,E1 122.260} C_DIS
LIN {X 0.073,Y -522.142,Z 667.475,A 0.000,B 0.000,C 90.000,E1 121.544} C_DIS
LIN {X -0.052,Y -525.940,Z 667.473,A 0.000,B 0.000,C 90.000,E1 121.131} C_DIS
LIN {X 0.195,Y -529.640,Z 667.471,A 0.000,B 0.000,C 90.000,E1 120.669} C_DIS
LIN {X -0.144,Y -534.063,Z 667.467,A 0.000,B 0.000,C 90.000,E1 120.129} C_DIS
LIN {X 0.009,Y -538.137,Z 667.464,A 0.000,B 0.000,C 90.000,E1 119.539} C_DIS
LIN {X 0.060,Y -542.610,Z 667.460,A 0.000,B 0.000,C 90.000,E1 118.821} C_DIS
LIN {X 0.155,Y -546.626,Z 667.456,A 0.000,B 0.000,C 90.000,E1 118.103} C_DIS
LIN {X -0.157,Y -550.264,Z 667.452,A 0.000,B 0.000,C 90.000,E1 117.436} C_DIS
LIN {X 0.020,Y -554.830,Z 667.447,A 0.000,B 0.000,C 90.000,E1 116.437} C_DIS
LIN {X -0.065,Y -556.713,Z 667.445,A 0.000,B 0.000,C 90.000,E1 116.027} C_DIS
LIN {X -0.205,Y -560.155,Z 667.440,A 0.000,B 0.000,C 90.000,E1 115.207} C_DIS
LIN {X 0.005,Y -564.282,Z 667.434,A 0.000,B 0.000,C 90.000,E1 114.079} C_DIS
LIN {X 0.278,Y -567.917,Z 667.428,A 0.000,B 0.000,C 90.000,E1 112.950} C_DIS
LIN {X 0.034,Y -570.397,Z 667.423,A 0.000,B 0.000,C 90.000,E1 112.153} C_DIS
LIN {X 0.206,Y -571.919,Z 667.420,A 0.000,B 0.000,C 90.000,E1 111.589} C_DIS
LIN {X -0.170,Y -574.489,Z 667.414,A 0.000,B 0.000,C 90.000,E1 110.536} C_DIS
LIN {X -0.176,Y -576.886,Z 667.408,A 0.000,B 0.000,C 90.000,E1 109.450} C_DIS
LIN {X 0.240,Y -579.643,Z 667.401,A 0.000,B 0.000,C 90.000,E1 108.055} C_DIS
LIN {X 0.189,Y -582.935,Z 667.391,A 0.000,B 0.000,C 90.000,E1 106.441} C_DIS
LIN {X -0.184,Y -585.594,Z 667.384,A 0.000,B 0.000,C 90.000,E1 105.134} C_DIS
LIN {X -0.263,Y -588.744,Z 667.375,A 0.000,B 0.000,C 90.000,E1 103.536} C_DIS
LIN {X 0.332,Y -590.755,Z 667.369,A 0.000,B 0.000,C 90.000,E1 102.411} C_DIS
LIN {X 0.096,Y -593.735,Z 667.360,A 0.000,B 0.000,C 90.000,E1 100.838} C_DIS
LIN {X 0.226,Y -596.252,Z 667.353,A 0.000,B 0.000,C 90.000,E1 99.500} C_DIS
LIN {X -0.195,Y -598.585,Z 667.346,A 0.000,B 0.000,C 90.000,E1 98.219} C_DIS
LIN {X 0.224,Y -600.285,Z 667.340,A 0.000,B 0.000,C 90.000,E1 97.125} C_DIS
LIN {X -0.225,Y -602.295,Z 667.332,A 0.000,B 0.000,C 90.000,E1 95.853} C_DIS
LIN {X -0.109,Y -604.181,Z 667.325,A 0.000,B 0.000,C 90.000,E1 94.531} C_DIS
LIN {X 0.001,Y -605.823,Z 667.318,A 0.000,B 0.000,C 90.000,E1 93.212} C_DIS
LIN {X -0.122,Y -606.970,Z 667.312,A 0.000,B 0.000,C 90.000,E1 92.178} C_DIS
LIN {X -0.236,Y -607.992,Z 667.306,A 0.000,B 0.000,C 90.000,E1 91.146} C_DIS
LIN {X -0.021,Y -608.565,Z 667.302,A 0.000,B 0.000,C 90.000,E1 90.344} C_DIS
LIN {X -0.130,Y -609.210,Z 667.296,A 0.000,B 0.000,C 90.000,E1 89.312} C_DIS
LIN {X -0.234,Y -609.580,Z 667.290,A 0.000,B 0.000,C 90.000,E1 88.282} C_DIS
LIN {X 0.293,Y -609.915,Z 667.285,A 0.000,B 0.000,C 90.000,E1 87.192} C_DIS
LIN {X -0.074,Y -610.055,Z 667.277,A 0.000,B 0.000,C 90.000,E1 85.927} C_DIS
LIN {X 0.190,Y -609.947,Z 667.273,A 0.000,B 0.000,C 90.000,E1 85.122} C_DIS
LIN {X -0.168,Y -609.681,Z 667.266,A 0.000,B 0.000,C 90.000,E1 83.856} C_DIS
LIN {X 0.062,Y -609.117,Z 667.259,A 0.000,B 0.000,C 90.000,E1 82.534} C_DIS
LIN {X -0.229,Y -608.735,Z 667.254,A 0.000,B 0.000,C 90.000,E1 81.781} C_DIS
LIN {X -0.188,Y -607.917,Z 667.248,A 0.000,B 0.000,C 90.000,E1 80.735} C_DIS
LIN {X 0.174,Y -606.566,Z 667.241,A 0.000,B 0.000,C 90.000,E1 79.398} C_DIS
LIN {X -0.028,Y -605.654,Z 667.237,A 0.000,B 0.000,C 90.000,E1 78.634} C_DIS
LIN {X -0.036,Y -604.379,Z 667.231,A 0.000,B 0.000,C 90.000,E1 77.589} C_DIS
LIN {X -0.074,Y -602.583,Z 667.224,A 0.000,B 0.000,C 90.000,E1 76.284} C_DIS
LIN {X -0.003,Y -601.016,Z 667.218,A 0.000,B 0.000,C 90.000,E1 75.227} C_DIS
LIN {X 0.194,Y -599.408,Z 667.212,A 0.000,B 0.000,C 90.000,E1 74.157} C_DIS
LIN {X -0.044,Y -596.736,Z 667.203,A 0.000,B 0.000,C 90.000,E1 72.598} C_DIS
LIN {X -0.033,Y -594.284,Z 667.196,A 0.000,B 0.000,C 90.000,E1 71.275} C_DIS
LIN {X 0.125,Y -591.593,Z 667.189,A 0.000,B 0.000,C 90.000,E1 69.934} C_DIS
LIN {X -0.198,Y -589.115,Z 667.183,A 0.000,B 0.000,C 90.000,E1 68.901} C_DIS
LIN {X 0.201,Y -586.459,Z 667.177,A 0.000,B 0.000,C 90.000,E1 67.794} C_DIS
LIN {X 0.015,Y -583.257,Z 667.171,A 0.000,B 0.000,C 90.000,E1 66.741} C_DIS
LIN {X -0.245,Y -581.621,Z 667.168,A 0.000,B 0.000,C 90.000,E1 66.230} C_DIS
LIN {X -0.116,Y -578.903,Z 667.163,A 0.000,B 0.000,C 90.000,E1 65.409} C_DIS
LIN {X -0.018,Y -576.014,Z 667.159,A 0.000,B 0.000,C 90.000,E1 64.588} C_DIS
LIN {X -0.110,Y -571.811,Z 667.153,A 0.000,B 0.000,C 90.000,E1 63.512} C_DIS
LIN {X 0.166,Y -568.483,Z 667.148,A 0.000,B 0.000,C 90.000,E1 62.666} C_DIS
LIN {X 0.231,Y -565.491,Z 667.144,A 0.000,B 0.000,C 90.000,E1 61.975} C_DIS
LIN {X 0.031,Y -562.262,Z 667.141,A 0.000,B 0.000,C 90.000,E1 61.307} C_DIS
LIN {X 0.297,Y -558.698,Z 667.137,A 0.000,B 0.000,C 90.000,E1 60.589} C_DIS
LIN {X 0.047,Y -554.582,Z 667.133,A 0.000,B 0.000,C 90.000,E1 59.921} C_DIS
LIN {X 0.354,Y -550.985,Z 667.130,A 0.000,B 0.000,C 90.000,E1 59.331} C_DIS
LIN {X 0.161,Y -546.974,Z 667.127,A 0.000,B 0.000,C 90.000,E1 58.791} C_DIS
LIN {X -0.057,Y -542.693,Z 667.124,A 0.000,B 0.000,C 90.000,E1 58.250} C_DIS
LIN {X 0.153,Y -537.931,Z 667.120,A 0.000,B 0.000,C 90.000,E1 57.661} C_DIS
LIN {X 0.025,Y -532.514,Z 667.117,A 0.000,B 0.000,C 90.000,E1 57.120} C_DIS
LIN {X -0.267,Y -526.608,Z 667.115,A 0.000,B 0.000,C 90.000,E1 56.628} C_DIS
LIN {X 0.155,Y -522.112,Z 667.112,A 0.000,B 0.000,C 90.000,E1 56.215} C_DIS
LIN {X 0.119,Y -517.344,Z 667.111,A 0.000,B 0.000,C 90.000,E1 55.881} C_DIS
LIN {X 0.170,Y -511.100,Z 667.108,A 0.000,B 0.000,C 90.000,E1 55.468} C_DIS
LIN {X 0.148,Y -502.779,Z 667.106,A 0.000,B 0.000,C 90.000,E1 54.975} C_DIS
LIN {X -0.042,Y -494.370,Z 667.103,A 0.000,B 0.000,C 90.000,E1 54.529} C_DIS
LIN {X -0.017,Y -477.666,Z 667.098,A 0.000,B 0.000,C 90.000,E1 53.623} C_DIS
LIN {X 0.035,Y -459.329,Z 667.092,A 0.000,B 0.000,C 90.000,E1 52.603} C_DIS
LIN {X -0.063,Y -436.028,Z 667.085,A 0.000,B 0.000,C 90.000,E1 51.251} C_DIS
LIN {X 0.067,Y -431.839,Z 667.083,A 0.000,B 0.000,C 90.000,E1 50.964} C_DIS
LIN {X 0.024,Y -431.784,Z 667.083,A 0.000,B 0.000,C 90.000,E1 50.964} C_DIS
LIN {X -0.142,Y -431.033,Z 667.081,A 0.000,B 0.000,C 90.000,E1 50.642} C_DIS
LIN {X -0.143,Y -421.901,Z 667.059,A 0.000,B 0.000,C 90.000,E1 46.620} C_DIS
LIN {X -0.077,Y -418.794,Z 667.050,A 0.000,B 0.000,C 90.000,E1 44.919} C_DIS
LIN {X 0.017,Y -417.410,Z 667.046,A 0.000,B 0.000,C 90.000,E1 44.312} C_DIS
LIN {X 0.008,Y -417.481,Z 667.032,A 0.000,B 0.000,C 90.000,E1 41.757} C_DIS
LIN {X -0.209,Y -418.186,Z 667.013,A 0.000,B 0.000,C 90.000,E1 38.382} C_DIS
LIN {X 0.072,Y -419.840,Z 666.994,A 0.000,B 0.000,C 90.000,E1 34.945} C_DIS
LIN {X 0.067,Y -420.806,Z 666.983,A 0.000,B 0.000,C 90.000,E1 32.911} C_DIS
LIN {X 0.097,Y -421.890,Z 666.972,A 0.000,B 0.000,C 90.000,E1 30.875} C_DIS
LIN {X -0.020,Y -422.634,Z 666.964,A 0.000,B 0.000,C 90.000,E1 29.539} C_DIS
LIN {X 0.109,Y -424.235,Z 666.949,A 0.000,B 0.000,C 90.000,E1 26.821} C_DIS
LIN {X -0.055,Y -425.596,Z 666.938,A 0.000,B 0.000,C 90.000,E1 24.823} C_DIS
LIN {X 0.184,Y -428.213,Z 666.921,A 0.000,B 0.000,C 90.000,E1 21.770} C_DIS
LIN {X 0.008,Y -429.766,Z 666.912,A 0.000,B 0.000,C 90.000,E1 20.120} C_DIS
LIN {X -0.165,Y -430.579,Z 666.906,A 0.000,B 0.000,C 90.000,E1 19.141} C_DIS
LIN {X -0.031,Y -431.724,Z 666.897,A 0.000,B 0.000,C 90.000,E1 17.457} C_DIS
LIN {X -0.189,Y -433.187,Z 666.886,A 0.000,B 0.000,C 90.000,E1 15.481} C_DIS
LIN {X -0.017,Y -434.914,Z 666.875,A 0.000,B 0.000,C 90.000,E1 13.467} C_DIS
LIN {X 0.000,Y -436.854,Z 666.864,A 0.000,B 0.000,C 90.000,E1 11.478} C_DIS
LIN {X 0.000,Y -439.980,Z 666.847,A 0.000,B 0.000,C 90.000,E1 8.511} C_DIS
LIN {X -0.189,Y -443.077,Z 666.833,A 0.000,B 0.000,C 90.000,E1 5.910} C_DIS
LIN {X 0.196,Y -446.985,Z 666.816,A 0.000,B 0.000,C 90.000,E1 2.922} C_DIS
LIN {X -0.097,Y -450.235,Z 666.804,A 0.000,B 0.000,C 90.000,E1 0.688} C_DIS
LIN {X 0.116,Y -454.362,Z 666.790,A 0.000,B 0.000,C 90.000,E1 358.165} C_DIS
LIN {X 0.055,Y -458.308,Z 666.777,A 0.000,B 0.000,C 90.000,E1 355.927} C_DIS
LIN {X 0.156,Y -461.257,Z 666.769,A 0.000,B 0.000,C 90.000,E1 354.318} C_DIS
LIN {X -0.107,Y -464.154,Z 666.760,A 0.000,B 0.000,C 90.000,E1 352.761} C_DIS
LIN {X 0.206,Y -467.074,Z 666.751,A 0.000,B 0.000,C 90.000,E1 351.141} C_DIS
LIN {X -0.076,Y -470.490,Z 666.740,A 0.000,B 0.000,C 90.000,E1 349.285} C_DIS
LIN {X 0.183,Y -474.365,Z 666.728,A 0.000,B 0.000,C 90.000,E1 347.061} C_DIS
LIN {X -0.111,Y -477.774,Z 666.718,A 0.000,B 0.000,C 90.000,E1 345.227} C_DIS
LIN {X -0.181,Y -480.706,Z 666.709,A 0.000,B 0.000,C 90.000,E1 343.685} C_DIS
LIN {X -0.210,Y -485.516,Z 666.696,A 0.000,B 0.000,C 90.000,E1 341.221} C_DIS
LIN {X 0.152,Y -488.569,Z 666.687,A 0.000,B 0.000,C 90.000,E1 339.645} C_DIS
LIN {X -0.168,Y -491.649,Z 666.679,A 0.000,B 0.000,C 90.000,E1 338.156} C_DIS
LIN {X -0.014,Y -494.003,Z 666.672,A 0.000,B 0.000,C 90.000,E1 336.922} C_DIS
LIN {X -0.081,Y -496.281,Z 666.665,A 0.000,B 0.000,C 90.000,E1 335.717} C_DIS
LIN {X 0.016,Y -501.816,Z 666.648,A 0.000,B 0.000,C 90.000,E1 332.692} C_DIS
LIN {X -0.075,Y -503.206,Z 666.645,A 0.000,B 0.000,C 90.000,E1 332.103} C_DIS
LIN {X -0.155,Y -504.984,Z 666.642,A 0.000,B 0.000,C 90.000,E1 331.513} C_DIS
LIN {X -0.033,Y -506.756,Z 666.639,A 0.000,B 0.000,C 90.000,E1 331.051} C_DIS
LIN {X 0.150,Y -508.536,Z 666.637,A 0.000,B 0.000,C 90.000,E1 330.717} C_DIS
LIN {X 0.044,Y -511.863,Z 666.635,A 0.000,B 0.000,C 90.000,E1 330.284} C_DIS
LIN {X -0.188,Y -516.600,Z 666.633,A 0.000,B 0.000,C 90.000,E1 329.871} C_DIS
LIN {X -0.052,Y -522.157,Z 666.630,A 0.000,B 0.000,C 90.000,E1 329.410} C_DIS
LIN {X 0.134,Y -533.027,Z 666.626,A 0.000,B 0.000,C 90.000,E1 328.614} C_DIS
LIN {X -0.011,Y -540.420,Z 666.623,A 0.000,B 0.000,C 90.000,E1 328.074} C_DIS
LIN {X 0.291,Y -546.192,Z 666.620,A 0.000,B 0.000,C 90.000,E1 327.582} C_DIS
LIN {X -0.245,Y -554.627,Z 666.616,A 0.000,B 0.000,C 90.000,E1 326.914} C_DIS
LIN {X 0.090,Y -562.811,Z 666.612,A 0.000,B 0.000,C 90.000,E1 326.135} C_DIS
LIN {X -0.047,Y -568.027,Z 666.609,A 0.000,B 0.000,C 90.000,E1 325.642} C_DIS
LIN {X -0.054,Y -574.465,Z 666.606,A 0.000,B 0.000,C 90.000,E1 325.022} C_DIS
LIN {X -0.297,Y -582.325,Z 666.601,A 0.000,B 0.000,C 90.000,E1 324.276} C_DIS
LIN {X 0.280,Y -591.156,Z 666.596,A 0.000,B 0.000,C 90.000,E1 323.336} C_DIS
LIN {X -0.071,Y -599.684,Z 666.592,A 0.000,B 0.000,C 90.000,E1 322.477} C_DIS
LIN {X -0.083,Y -605.625,Z 666.588,A 0.000,B 0.000,C 90.000,E1 321.823} C_DIS
LIN {X -0.080,Y -611.241,Z 666.584,A 0.000,B 0.000,C 90.000,E1 321.170} C_DIS
LIN {X -0.030,Y -616.451,Z 666.581,A 0.000,B 0.000,C 90.000,E1 320.517} C_DIS
LIN {X -0.056,Y -622.379,Z 666.576,A 0.000,B 0.000,C 90.000,E1 319.747} C_DIS
LIN {X 0.325,Y -629.502,Z 666.571,A 0.000,B 0.000,C 90.000,E1 318.690} C_DIS
LIN {X 0.016,Y -634.477,Z 666.566,A 0.000,B 0.000,C 90.000,E1 317.957} C_DIS
LIN {X 0.110,Y -640.020,Z 666.562,A 0.000,B 0.000,C 90.000,E1 317.067} C_DIS
LIN {X 0.255,Y -646.009,Z 666.556,A 0.000,B 0.000,C 90.000,E1 316.053} C_DIS
LIN {X -0.037,Y -653.084,Z 666.549,A 0.000,B 0.000,C 90.000,E1 314.838} C_DIS
LIN {X -0.160,Y -657.111,Z 666.545,A 0.000,B 0.000,C 90.000,E1 314.109} C_DIS
LIN {X 0.196,Y -663.241,Z 666.538,A 0.000,B 0.000,C 90.000,E1 312.852} C_DIS
LIN {X -0.292,Y -667.884,Z 666.533,A 0.000,B 0.000,C 90.000,E1 311.919} C_DIS
LIN {X 0.215,Y -672.381,Z 666.527,A 0.000,B 0.000,C 90.000,E1 310.906} C_DIS
LIN {X 0.339,Y -676.418,Z 666.522,A 0.000,B 0.000,C 90.000,E1 309.930} C_DIS
LIN {X -0.056,Y -678.321,Z 666.519,A 0.000,B 0.000,C 90.000,E1 309.483} C_DIS
LIN {X 0.112,Y -680.885,Z 666.515,A 0.000,B 0.000,C 90.000,E1 308.749} C_DIS
LIN {X -0.081,Y -684.064,Z 666.510,A 0.000,B 0.000,C 90.000,E1 307.810} C_DIS
LIN {X 0.143,Y -686.182,Z 666.506,A 0.000,B 0.000,C 90.000,E1 307.076} C_DIS
LIN {X 0.199,Y -689.412,Z 666.500,A 0.000,B 0.000,C 90.000,E1 305.884} C_DIS
LIN {X 0.105,Y -691.765,Z 666.494,A 0.000,B 0.000,C 90.000,E1 304.945} C_DIS
LIN {X -0.143,Y -694.385,Z 666.488,A 0.000,B 0.000,C 90.000,E1 303.785} C_DIS
LIN {X 0.003,Y -696.271,Z 666.482,A 0.000,B 0.000,C 90.000,E1 302.832} C_DIS
LIN {X -0.073,Y -697.514,Z 666.479,A 0.000,B 0.000,C 90.000,E1 302.133} C_DIS
LIN {X 0.361,Y -699.407,Z 666.472,A 0.000,B 0.000,C 90.000,E1 300.924} C_DIS
LIN {X -0.061,Y -700.374,Z 666.468,A 0.000,B 0.000,C 90.000,E1 300.256} C_DIS
LIN {X -0.136,Y -700.998,Z 666.466,A 0.000,B 0.000,C 90.000,E1 299.795} C_DIS
LIN {X 0.000,Y -702.225,Z 666.459,A 0.000,B 0.000,C 90.000,E1 298.615} C_DIS
LIN {X -0.174,Y -703.354,Z 666.453,A 0.000,B 0.000,C 90.000,E1 297.462} C_DIS
LIN {X -0.010,Y -704.408,Z 666.446,A 0.000,B 0.000,C 90.000,E1 296.283} C_DIS
LIN {X -0.094,Y -704.787,Z 666.442,A 0.000,B 0.000,C 90.000,E1 295.591} C_DIS
LIN {X 0.182,Y -704.246,Z 666.440,A 0.000,B 0.000,C 90.000,E1 295.103} C_DIS
LIN {X -0.171,Y -703.806,Z 666.438,A 0.000,B 0.000,C 90.000,E1 294.899} C_DIS
LIN {X 0.255,Y -702.082,Z 666.436,A 0.000,B 0.000,C 90.000,E1 294.515} C_DIS
LIN {X -0.394,Y -700.812,Z 666.435,A 0.000,B 0.000,C 90.000,E1 294.335} C_DIS
LIN {X -0.256,Y -699.947,Z 666.434,A 0.000,B 0.000,C 90.000,E1 294.207} C_DIS
LIN {X -0.120,Y -698.658,Z 666.434,A 0.000,B 0.000,C 90.000,E1 294.079} C_DIS
LIN {X 0.387,Y -695.421,Z 666.433,A 0.000,B 0.000,C 90.000,E1 293.823} C_DIS
LIN {X 0.302,Y -692.356,Z 666.432,A 0.000,B 0.000,C 90.000,E1 293.643} C_DIS
LIN {X 0.126,Y -690.426,Z 666.431,A 0.000,B 0.000,C 90.000,E1 293.567} C_DIS
LIN {X -0.144,Y -687.864,Z 666.431,A 0.000,B 0.000,C 90.000,E1 293.515} C_DIS
LIN {X 0.187,Y -680.656,Z 666.430,A 0.000,B 0.000,C 90.000,E1 293.334} C_DIS
LIN {X 0.299,Y -671.342,Z 666.429,A 0.000,B 0.000,C 90.000,E1 293.206} C_DIS
LIN {X -0.047,Y -663.295,Z 666.429,A 0.000,B 0.000,C 90.000,E1 293.153} C_DIS
LIN {X -0.164,Y -653.529,Z 666.428,A 0.000,B 0.000,C 90.000,E1 293.025} C_DIS
LIN {X 0.165,Y -643.551,Z 666.427,A 0.000,B 0.000,C 90.000,E1 292.823} C_DIS
LIN {X -0.107,Y -633.611,Z 666.426,A 0.000,B 0.000,C 90.000,E1 292.642} C_DIS
LIN {X -0.271,Y -620.278,Z 666.424,A 0.000,B 0.000,C 90.000,E1 292.333} C_DIS
LIN {X 0.343,Y -606.817,Z 666.422,A 0.000,B 0.000,C 90.000,E1 291.897} C_DIS
LIN {X 0.211,Y -579.145,Z 666.417,A 0.000,B 0.000,C 90.000,E1 291.046} C_DIS
LIN {X 0.084,Y -563.360,Z 666.415,A 0.000,B 0.000,C 90.000,E1 290.610} C_DIS
LIN {X 0.181,Y -556.928,Z 666.413,A 0.000,B 0.000,C 90.000,E1 290.301} C_DIS
LIN {X -0.144,Y -556.263,Z 666.413,A 0.000,B 0.000,C 90.000,E1 290.301} C_DIS
LIN {X -0.190,Y -556.216,Z 666.413,A 0.000,B 0.000,C 90.000,E1 290.301} C_DIS
LIN {X 0.149,Y -555.235,Z 666.412,A 0.000,B 0.000,C 90.000,E1 290.120} C_DIS
LIN {X 0.107,Y -555.216,Z 666.412,A 0.000,B 0.000,C 90.000,E1 290.120} C_DIS
LIN {X 0.168,Y -554.634,Z 666.409,A 0.000,B 0.000,C 90.000,E1 289.631} C_DIS
LIN {X 0.312,Y -554.394,Z 666.405,A 0.000,B 0.000,C 90.000,E1 288.779} C_DIS
LIN {X 0.029,Y -554.242,Z 666.398,A 0.000,B 0.000,C 90.000,E1 287.692} C_DIS
LIN {X -0.149,Y -553.844,Z 666.391,A 0.000,B 0.000,C 90.000,E1 286.315} C_DIS
LIN {X 0.312,Y -553.250,Z 666.381,A 0.000,B 0.000,C 90.000,E1 284.592} C_DIS
LIN {X -0.284,Y -552.668,Z 666.375,A 0.000,B 0.000,C 90.000,E1 283.536} C_DIS
LIN {X 0.131,Y -551.650,Z 666.364,A 0.000,B 0.000,C 90.000,E1 281.535} C_DIS
LIN {X -0.247,Y -550.741,Z 666.353,A 0.000,B 0.000,C 90.000,E1 279.613} C_DIS
LIN {X -0.187,Y -550.160,Z 666.342,A 0.000,B 0.000,C 90.000,E1 277.644} C_DIS
LIN {X 0.294,Y -549.806,Z 666.333,A 0.000,B 0.000,C 90.000,E1 275.910} C_DIS
LIN {X 0.244,Y -549.562,Z 666.321,A 0.000,B 0.000,C 90.000,E1 273.669} C_DIS
LIN {X -0.074,Y -549.337,Z 666.314,A 0.000,B 0.000,C 90.000,E1 272.579} C_DIS
LIN {X 0.152,Y -549.016,Z 666.308,A 0.000,B 0.000,C 90.000,E1 271.432} C_DIS
LIN {X -0.139,Y -548.384,Z 666.300,A 0.000,B 0.000,C 90.000,E1 270.057} C_DIS
LIN {X 0.106,Y -547.624,Z 666.292,A 0.000,B 0.000,C 90.000,E1 268.625} C_DIS
LIN {X -0.242,Y -546.992,Z 666.286,A 0.000,B 0.000,C 90.000,E1 267.535} C_DIS
LIN {X -0.011,Y -546.168,Z 666.278,A 0.000,B 0.000,C 90.000,E1 266.102} C_DIS
LIN {X 0.235,Y -545.094,Z 666.271,A 0.000,B 0.000,C 90.000,E1 264.666} C_DIS
LIN {X -0.026,Y -543.869,Z 666.263,A 0.000,B 0.000,C 90.000,E1 263.280} C_DIS
LIN {X -0.145,Y -541.801,Z 666.252,A 0.000,B 0.000,C 90.000,E1 261.310} C_DIS
LIN {X -0.106,Y -539.062,Z 666.236,A 0.000,B 0.000,C 90.000,E1 258.465} C_DIS
LIN {X -0.045,Y -537.410,Z 666.225,A 0.000,B 0.000,C 90.000,E1 256.464} C_DIS
LIN {X -0.137,Y -536.199,Z 666.217,A 0.000,B 0.000,C 90.000,E1 255.046} C_DIS
LIN {X -0.109,Y -534.831,Z 666.209,A 0.000,B 0.000,C 90.000,E1 253.614} C_DIS
LIN {X -0.109,Y -533.381,Z 666.201,A 0.000,B 0.000,C 90.000,E1 252.181} C_DIS
LIN {X 0.022,Y -532.004,Z 666.193,A 0.000,B 0.000,C 90.000,E1 250.732} C_DIS
LIN {X 0.115,Y -530.688,Z 666.187,A 0.000,B 0.000,C 90.000,E1 249.571} C_DIS
LIN {X 0.063,Y -528.260,Z 666.177,A 0.000,B 0.000,C 90.000,E1 247.847} C_DIS
LIN {X 0.294,Y -526.639,Z 666.171,A 0.000,B 0.000,C 90.000,E1 246.666} C_DIS
LIN {X 0.160,Y -525.710,Z 666.167,A 0.000,B 0.000,C 90.000,E1 246.102} C_DIS
LIN {X -0.286,Y -522.657,Z 666.158,A 0.000,B 0.000,C 90.000,E1 244.409} C_DIS
LIN {X -0.075,Y -521.020,Z 666.153,A 0.000,B 0.000,C 90.000,E1 243.512} C_DIS
LIN {X 0.162,Y -518.108,Z 666.145,A 0.000,B 0.000,C 90.000,E1 242.025} C_DIS
LIN {X -0.112,Y -515.081,Z 666.137,A 0.000,B 0.000,C 90.000,E1 240.589} C_DIS
LIN {X -0.186,Y -511.840,Z 666.128,A 0.000,B 0.000,C 90.000,E1 239.125} C_DIS
LIN {X -0.320,Y -508.560,Z 666.120,A 0.000,B 0.000,C 90.000,E1 237.661} C_DIS
LIN {X 0.341,Y -504.481,Z 666.110,A 0.000,B 0.000,C 90.000,E1 235.801} C_DIS
LIN {X 0.024,Y -501.513,Z 666.104,A 0.000,B 0.000,C 90.000,E1 234.642} C_DIS
LIN {X 0.116,Y -497.715,Z 666.095,A 0.000,B 0.000,C 90.000,E1 233.130} C_DIS
LIN {X 0.016,Y -491.822,Z 666.082,A 0.000,B 0.000,C 90.000,E1 230.723} C_DIS
LIN {X -0.305,Y -487.483,Z 666.072,A 0.000,B 0.000,C 90.000,E1 228.933} C_DIS
LIN {X -0.079,Y -483.083,Z 666.061,A 0.000,B 0.000,C 90.000,E1 227.067} C_DIS
LIN {X 0.249,Y -479.461,Z 666.053,A 0.000,B 0.000,C 90.000,E1 225.486} C_DIS
LIN {X 0.051,Y -476.506,Z 666.046,A 0.000,B 0.000,C 90.000,E1 224.271} C_DIS
LIN {X 0.250,Y -472.880,Z 666.037,A 0.000,B 0.000,C 90.000,E1 222.690} C_DIS
LIN {X 0.092,Y -466.652,Z 666.022,A 0.000,B 0.000,C 90.000,E1 219.886} C_DIS
LIN {X 0.132,Y -463.428,Z 666.013,A 0.000,B 0.000,C 90.000,E1 218.302} C_DIS
LIN {X 0.030,Y -458.916,Z 666.001,A 0.000,B 0.000,C 90.000,E1 216.091} C_DIS
LIN {X -0.179,Y -455.201,Z 665.990,A 0.000,B 0.000,C 90.000,E1 214.199} C_DIS
LIN {X 0.187,Y -452.172,Z 665.981,A 0.000,B 0.000,C 90.000,E1 212.546} C_DIS
LIN {X -0.291,Y -448.579,Z 665.970,A 0.000,B 0.000,C 90.000,E1 210.669} C_DIS
LIN {X -0.074,Y -445.018,Z 665.959,A 0.000,B 0.000,C 90.000,E1 208.693} C_DIS
LIN {X -0.157,Y -441.504,Z 665.949,A 0.000,B 0.000,C 90.000,E1 206.744} C_DIS
LIN {X -0.129,Y -438.002,Z 665.938,A 0.000,B 0.000,C 90.000,E1 204.771} C_DIS
LIN {X 0.199,Y -435.004,Z 665.928,A 0.000,B 0.000,C 90.000,E1 203.078} C_DIS
LIN {X -0.107,Y -431.996,Z 665.919,A 0.000,B 0.000,C 90.000,E1 201.461} C_DIS
LIN {X -0.016,Y -428.388,Z 665.908,A 0.000,B 0.000,C 90.000,E1 199.450} C_DIS
LIN {X 0.046,Y -424.434,Z 665.895,A 0.000,B 0.000,C 90.000,E1 197.094} C_DIS
LIN {X 0.094,Y -421.033,Z 665.884,A 0.000,B 0.000,C 90.000,E1 195.064} C_DIS
LIN {X 0.198,Y -418.209,Z 665.874,A 0.000,B 0.000,C 90.000,E1 193.355} C_DIS
LIN {X 0.021,Y -413.316,Z 665.857,A 0.000,B 0.000,C 90.000,E1 190.310} C_DIS
LIN {X -0.164,Y -410.199,Z 665.846,A 0.000,B 0.000,C 90.000,E1 188.276} C_DIS
LIN {X -0.098,Y -407.612,Z 665.836,A 0.000,B 0.000,C 90.000,E1 186.543} C_DIS
LIN {X 0.165,Y -403.438,Z 665.819,A 0.000,B 0.000,C 90.000,E1 183.383} C_DIS
LIN {X -0.067,Y -400.620,Z 665.805,A 0.000,B 0.000,C 90.000,E1 180.974} C_DIS
LIN {X 0.152,Y -396.917,Z 665.782,A 0.000,B 0.000,C 90.000,E1 176.731} C_DIS
LIN {X 0.136,Y -395.205,Z 665.766,A 0.000,B 0.000,C 90.000,E1 173.913} C_DIS
LIN {X -0.172,Y -394.351,Z 665.755,A 0.000,B 0.000,C 90.000,E1 171.837} C_DIS
LIN {X -0.086,Y -393.491,Z 665.735,A 0.000,B 0.000,C 90.000,E1 168.285} C_DIS
LIN {X -0.171,Y -393.296,Z 665.723,A 0.000,B 0.000,C 90.000,E1 166.172} C_DIS
LIN {X -0.019,Y -393.292,Z 665.705,A 0.000,B 0.000,C 90.000,E1 162.960} C_DIS
LIN {X -0.131,Y -393.604,Z 665.692,A 0.000,B 0.000,C 90.000,E1 160.496} C_DIS
LIN {X 0.169,Y -393.731,Z 665.686,A 0.000,B 0.000,C 90.000,E1 159.390} C_DIS
LIN {X 0.101,Y -394.090,Z 665.672,A 0.000,B 0.000,C 90.000,E1 156.922} C_DIS
LIN {X -0.003,Y -394.510,Z 665.658,A 0.000,B 0.000,C 90.000,E1 154.460} C_DIS
LIN {X -0.003,Y -394.892,Z 665.648,A 0.000,B 0.000,C 90.000,E1 152.692} C_DIS
LIN {X -0.120,Y -395.363,Z 665.637,A 0.000,B 0.000,C 90.000,E1 150.589} C_DIS
LIN {X 0.109,Y -395.824,Z 665.627,A 0.000,B 0.000,C 90.000,E1 148.791} C_DIS
LIN {X -0.032,Y -396.628,Z 665.613,A 0.000,B 0.000,C 90.000,E1 146.342} C_DIS
LIN {X 0.059,Y -397.737,Z 665.599,A 0.000,B 0.000,C 90.000,E1 143.863} C_DIS
LIN {X -0.006,Y -399.007,Z 665.586,A 0.000,B 0.000,C 90.000,E1 141.412} C_DIS
LIN {X 0.161,Y -400.601,Z 665.572,A 0.000,B 0.000,C 90.000,E1 138.933} C_DIS
LIN {X -0.162,Y -401.669,Z 665.562,A 0.000,B 0.000,C 90.000,E1 137.229} C_DIS
LIN {X 0.260,Y -403.915,Z 665.545,A 0.000,B 0.000,C 90.000,E1 134.028} C_DIS
LIN {X -0.082,Y -404.512,Z 665.541,A 0.000,B 0.000,C 90.000,E1 133.380} C_DIS
LIN {X -0.210,Y -405.748,Z 665.536,A 0.000,B 0.000,C 90.000,E1 132.528} C_DIS
LIN {X 0.005,Y -406.226,Z 665.535,A 0.000,B 0.000,C 90.000,E1 132.324} C_DIS
LIN {X 0.021,Y -407.484,Z 665.532,A 0.000,B 0.000,C 90.000,E1 131.714} C_DIS
LIN {X -0.100,Y -408.713,Z 665.530,A 0.000,B 0.000,C 90.000,E1 131.472} C_DIS
LIN {X -0.220,Y -409.700,Z 665.529,A 0.000,B 0.000,C 90.000,E1 131.229} C_DIS
LIN {X -0.145,Y -413.298,Z 665.526,A 0.000,B 0.000,C 90.000,E1 130.701} C_DIS
LIN {X 0.020,Y -417.119,Z 665.524,A 0.000,B 0.000,C 90.000,E1 130.297} C_DIS
LIN {X -0.156,Y -423.149,Z 665.521,A 0.000,B 0.000,C 90.000,E1 129.806} C_DIS
LIN {X -0.087,Y -451.379,Z 665.509,A 0.000,B 0.000,C 90.000,E1 127.649} C_DIS
LIN {X -0.118,Y -460.829,Z 665.505,A 0.000,B 0.000,C 90.000,E1 126.950} C_DIS
LIN {X -0.021,Y -469.904,Z 665.501,A 0.000,B 0.000,C 90.000,E1 126.251} C_DIS
LIN {X -0.001,Y -480.493,Z 665.497,A 0.000,B 0.000,C 90.000,E1 125.391} C_DIS
LIN {X 0.068,Y -487.622,Z 665.493,A 0.000,B 0.000,C 90.000,E1 124.771} C_DIS
LIN {X -0.119,Y -491.990,Z 665.491,A 0.000,B 0.000,C 90.000,E1 124.405} C_DIS
LIN {X -0.124,Y -500.526,Z 665.487,A 0.000,B 0.000,C 90.000,E1 123.627} C_DIS
LIN {X -0.052,Y -507.326,Z 665.483,A 0.000,B 0.000,C 90.000,E1 122.959} C_DIS
LIN {X -0.011,Y -511.432,Z 665.481,A 0.000,B 0.000,C 90.000,E1 122.546} C_DIS
LIN {X -0.105,Y -516.816,Z 665.478,A 0.000,B 0.000,C 90.000,E1 122.005} C_DIS
LIN {X -0.151,Y -520.735,Z 665.475,A 0.000,B 0.000,C 90.000,E1 121.592} C_DIS
LIN {X -0.072,Y -525.574,Z 665.473,A 0.000,B 0.000,C 90.000,E1 121.052} C_DIS
LIN {X 0.063,Y -528.138,Z 665.471,A 0.000,B 0.000,C 90.000,E1 120.747} C_DIS
LIN {X 0.095,Y -532.442,Z 665.468,A 0.000,B 0.000,C 90.000,E1 120.207} C_DIS
LIN {X 0.138,Y -537.360,Z 665.464,A 0.000,B 0.000,C 90.000,E1 119.539} C_DIS
LIN {X 0.142,Y -541.787,Z 665.461,A 0.000,B 0.000,C 90.000,E1 118.871} C_DIS
LIN {X 0.055,Y -545.929,Z 665.457,A 0.000,B 0.000,C 90.000,E1 118.180} C_DIS
LIN {X 0.180,Y -549.729,Z 665.453,A 0.000,B 0.000,C 90.000,E1 117.462} C_DIS
LIN {X 0.112,Y -554.399,Z 665.447,A 0.000,B 0.000,C 90.000,E1 116.488} C_DIS
LIN {X -0.221,Y -556.336,Z 665.445,A 0.000,B 0.000,C 90.000,E1 116.104} C_DIS
LIN {X -0.363,Y -559.831,Z 665.440,A 0.000,B 0.000,C 90.000,E1 115.283} C_DIS
LIN {X 0.077,Y -564.035,Z 665.434,A 0.000,B 0.000,C 90.000,E1 114.131} C_DIS
LIN {X 0.120,Y -567.758,Z 665.428,A 0.000,B 0.000,C 90.000,E1 113.025} C_DIS
LIN {X 0.095,Y -570.304,Z 665.423,A 0.000,B 0.000,C 90.000,E1 112.206} C_DIS
LIN {X 0.053,Y -571.899,Z 665.420,A 0.000,B 0.000,C 90.000,E1 111.663} C_DIS
LIN {X 0.220,Y -574.526,Z 665.414,A 0.000,B 0.000,C 90.000,E1 110.556} C_DIS
LIN {X -0.124,Y -576.988,Z 665.408,A 0.000,B 0.000,C 90.000,E1 109.504} C_DIS
LIN {X -0.090,Y -579.251,Z 665.402,A 0.000,B 0.000,C 90.000,E1 108.417} C_DIS
LIN {X 0.237,Y -583.128,Z 665.392,A 0.000,B 0.000,C 90.000,E1 106.496} C_DIS
LIN {X 0.104,Y -586.351,Z 665.383,A 0.000,B 0.000,C 90.000,E1 104.898} C_DIS
LIN {X -0.214,Y -589.007,Z 665.375,A 0.000,B 0.000,C 90.000,E1 103.592} C_DIS
LIN {X -0.322,Y -591.058,Z 665.370,A 0.000,B 0.000,C 90.000,E1 102.535} C_DIS
LIN {X -0.157,Y -594.612,Z 665.359,A 0.000,B 0.000,C 90.000,E1 100.658} C_DIS
LIN {X 0.284,Y -596.623,Z 665.353,A 0.000,B 0.000,C 90.000,E1 99.557} C_DIS
LIN {X 0.169,Y -598.564,Z 665.347,A 0.000,B 0.000,C 90.000,E1 98.511} C_DIS
LIN {X 0.072,Y -600.320,Z 665.342,A 0.000,B 0.000,C 90.000,E1 97.466} C_DIS
LIN {X 0.149,Y -602.420,Z 665.334,A 0.000,B 0.000,C 90.000,E1 96.144} C_DIS
LIN {X -0.027,Y -604.742,Z 665.326,A 0.000,B 0.000,C 90.000,E1 94.588} C_DIS
LIN {X 0.092,Y -606.393,Z 665.318,A 0.000,B 0.000,C 90.000,E1 93.269} C_DIS
LIN {X -0.024,Y -607.562,Z 665.312,A 0.000,B 0.000,C 90.000,E1 92.236} C_DIS
LIN {X -0.131,Y -608.593,Z 665.307,A 0.000,B 0.000,C 90.000,E1 91.203} C_DIS
LIN {X -0.239,Y -609.373,Z 665.301,A 0.000,B 0.000,C 90.000,E1 90.172} C_DIS
LIN {X 0.273,Y -609.961,Z 665.295,A 0.000,B 0.000,C 90.000,E1 89.083} C_DIS
LIN {X -0.130,Y -610.436,Z 665.288,A 0.000,B 0.000,C 90.000,E1 87.822} C_DIS
LIN {X -0.193,Y -610.644,Z 665.282,A 0.000,B 0.000,C 90.000,E1 86.788} C_DIS
LIN {X -0.253,Y -610.699,Z 665.276,A 0.000,B 0.000,C 90.000,E1 85.755} C_DIS
LIN {X 0.009,Y -610.463,Z 665.269,A 0.000,B 0.000,C 90.000,E1 84.432} C_DIS
LIN {X -0.004,Y -610.129,Z 665.263,A 0.000,B 0.000,C 90.000,E1 83.394} C_DIS
LIN {X 0.315,Y -609.522,Z 665.256,A 0.000,B 0.000,C 90.000,E1 82.064} C_DIS
LIN {X -0.057,Y -608.980,Z 665.252,A 0.000,B 0.000,C 90.000,E1 81.319} C_DIS
LIN {X -0.015,Y -608.012,Z 665.246,A 0.000,B 0.000,C 90.000,E1 80.274} C_DIS
LIN {X -0.254,Y -606.599,Z 665.239,A 0.000,B 0.000,C 90.000,E1 78.993} C_DIS
LIN {X -0.072,Y -604.604,Z 665.230,A 0.000,B 0.000,C 90.000,E1 77.409} C_DIS
LIN {X -0.245,Y -602.738,Z 665.223,A 0.000,B 0.000,C 90.000,E1 76.117} C_DIS
LIN {X -0.003,Y -600.332,Z 665.214,A 0.000,B 0.000,C 90.000,E1 74.519} C_DIS
LIN {X 0.179,Y -598.538,Z 665.208,A 0.000,B 0.000,C 90.000,E1 73.449} C_DIS
LIN {X -0.060,Y -596.671,Z 665.202,A 0.000,B 0.000,C 90.000,E1 72.417} C_DIS
LIN {X 0.063,Y -594.714,Z 665.196,A 0.000,B 0.000,C 90.000,E1 71.348} C_DIS
LIN {X 0.219,Y -591.973,Z 665.189,A 0.000,B 0.000,C 90.000,E1 70.007} C_DIS
LIN {X 0.222,Y -590.142,Z 665.185,A 0.000,B 0.000,C 90.000,E1 69.209} C_DIS
LIN {X -0.252,Y -586.748,Z 665.177,A 0.000,B 0.000,C 90.000,E1 67.922} C_DIS
LIN {X 0.333,Y -583.545,Z 665.171,A 0.000,B 0.000,C 90.000,E1 66.794} C_DIS
LIN {X -0.157,Y -581.879,Z 665.168,A 0.000,B 0.000,C 90.000,E1 66.305} C_DIS
LIN {X -0.032,Y -579.100,Z 665.164,A 0.000,B 0.000,C 90.000,E1 65.485} C_DIS
LIN {X -0.083,Y -575.138,Z 665.158,A 0.000,B 0.000,C 90.000,E1 64.409} C_DIS
LIN {X 0.065,Y -570.780,Z 665.152,A 0.000,B 0.000,C 90.000,E1 63.307} C_DIS
LIN {X 0.070,Y -567.340,Z 665.147,A 0.000,B 0.000,C 90.000,E1 62.487} C_DIS
LIN {X -0.285,Y -564.865,Z 665.144,A 0.000,B 0.000,C 90.000,E1 61.975} C_DIS
LIN {X 0.102,Y -562.250,Z 665.141,A 0.000,B 0.000,C 90.000,E1 61.385} C_DIS
LIN {X -0.123,Y -558.572,Z 665.137,A 0.000,B 0.000,C 90.000,E1 60.717} C_DIS
LIN {X 0.109,Y -554.404,Z 665.133,A 0.000,B 0.000,C 90.000,E1 59.999} C_DIS
LIN {X -0.108,Y -549.767,Z 665.130,A 0.000,B 0.000,C 90.000,E1 59.331} C_DIS
LIN {X 0.160,Y -545.634,Z 665.126,A 0.000,B 0.000,C 90.000,E1 58.742} C_DIS
LIN {X -0.070,Y -541.105,Z 665.123,A 0.000,B 0.000,C 90.000,E1 58.201} C_DIS
LIN {X 0.165,Y -536.558,Z 665.120,A 0.000,B 0.000,C 90.000,E1 57.661} C_DIS
LIN {X 0.137,Y -531.505,Z 665.118,A 0.000,B 0.000,C 90.000,E1 57.168} C_DIS
LIN {X 0.086,Y -526.098,Z 665.115,A 0.000,B 0.000,C 90.000,E1 56.707} C_DIS
LIN {X -0.247,Y -522.073,Z 665.113,A 0.000,B 0.000,C 90.000,E1 56.421} C_DIS
LIN {X 0.093,Y -515.602,Z 665.111,A 0.000,B 0.000,C 90.000,E1 55.928} C_DIS
LIN {X 0.084,Y -508.872,Z 665.109,A 0.000,B 0.000,C 90.000,E1 55.515} C_DIS
LIN {X 0.025,Y -502.272,Z 665.106,A 0.000,B 0.000,C 90.000,E1 55.135} C_DIS
LIN {X -0.037,Y -495.491,Z 665.104,A 0.000,B 0.000,C 90.000,E1 54.769} C_DIS
LIN {X -0.093,Y -477.086,Z 665.099,A 0.000,B 0.000,C 90.000,E1 53.783} C_DIS
LIN {X -0.014,Y -458.777,Z 665.093,A 0.000,B 0.000,C 90.000,E1 52.763} C_DIS
LIN {X 0.120,Y -435.910,Z 665.086,A 0.000,B 0.000,C 90.000,E1 51.412} C_DIS
LIN {X 0.137,Y -432.216,Z 665.084,A 0.000,B 0.000,C 90.000,E1 51.170} C_DIS
LIN {X 0.111,Y -432.174,Z 665.084,A 0.000,B 0.000,C 90.000,E1 51.170} C_DIS
LIN {X -0.212,Y -431.217,Z 665.082,A 0.000,B 0.000,C 90.000,E1 50.723} C_DIS
LIN {X 0.082,Y -422.043,Z 665.059,A 0.000,B 0.000,C 90.000,E1 46.662} C_DIS
LIN {X -0.138,Y -418.919,Z 665.050,A 0.000,B 0.000,C 90.000,E1 45.000} C_DIS
LIN {X -0.013,Y -417.794,Z 665.047,A 0.000,B 0.000,C 90.000,E1 44.474} C_DIS
LIN {X 0.124,Y -417.925,Z 665.035,A 0.000,B 0.000,C 90.000,E1 42.243} C_DIS
LIN {X -0.061,Y -418.272,Z 665.022,A 0.000,B 0.000,C 90.000,E1 39.886} C_DIS
LIN {X 0.210,Y -419.354,Z 665.005,A 0.000,B 0.000,C 90.000,E1 36.790} C_DIS
LIN {X 0.080,Y -420.455,Z 664.993,A 0.000,B 0.000,C 90.000,E1 34.771} C_DIS
LIN {X -0.056,Y -421.630,Z 664.980,A 0.000,B 0.000,C 90.000,E1 32.418} C_DIS
LIN {X 0.043,Y -422.351,Z 664.973,A 0.000,B 0.000,C 90.000,E1 31.052} C_DIS
LIN {X 0.060,Y -423.260,Z 664.963,A 0.000,B 0.000,C 90.000,E1 29.361} C_DIS
LIN {X 0.058,Y -424.650,Z 664.950,A 0.000,B 0.000,C 90.000,E1 27.001} C_DIS
LIN {X 0.077,Y -426.186,Z 664.937,A 0.000,B 0.000,C 90.000,E1 24.643} C_DIS
LIN {X -0.015,Y -428.536,Z 664.922,A 0.000,B 0.000,C 90.000,E1 21.972} C_DIS
LIN {X -0.028,Y -430.099,Z 664.913,A 0.000,B 0.000,C 90.000,E1 20.301} C_DIS
LIN {X 0.018,Y -431.110,Z 664.905,A 0.000,B 0.000,C 90.000,E1 18.960} C_DIS
LIN {X -0.154,Y -432.461,Z 664.894,A 0.000,B 0.000,C 90.000,E1 16.985} C_DIS
LIN {X 0.015,Y -433.670,Z 664.885,A 0.000,B 0.000,C 90.000,E1 15.300} C_DIS
LIN {X -0.027,Y -435.098,Z 664.876,A 0.000,B 0.000,C 90.000,E1 13.647} C_DIS
LIN {X -0.002,Y -437.002,Z 664.865,A 0.000,B 0.000,C 90.000,E1 11.658} C_DIS
LIN {X -0.070,Y -439.672,Z 664.850,A 0.000,B 0.000,C 90.000,E1 9.029} C_DIS
LIN {X 0.036,Y -441.122,Z 664.843,A 0.000,B 0.000,C 90.000,E1 7.701} C_DIS
LIN {X -0.162,Y -443.114,Z 664.834,A 0.000,B 0.000,C 90.000,E1 6.087} C_DIS
LIN {X -0.194,Y -445.559,Z 664.823,A 0.000,B 0.000,C 90.000,E1 4.131} C_DIS
LIN {X 0.102,Y -447.867,Z 664.814,A 0.000,B 0.000,C 90.000,E1 2.465} C_DIS
LIN {X 0.171,Y -451.813,Z 664.799,A 0.000,B 0.000,C 90.000,E1 359.771} C_DIS
LIN {X -0.160,Y -455.074,Z 664.788,A 0.000,B 0.000,C 90.000,E1 357.879} C_DIS
LIN {X -0.208,Y -459.034,Z 664.776,A 0.000,B 0.000,C 90.000,E1 355.641} C_DIS
LIN {X -0.102,Y -461.943,Z 664.767,A 0.000,B 0.000,C 90.000,E1 354.033} C_DIS
LIN {X 0.161,Y -464.838,Z 664.758,A 0.000,B 0.000,C 90.000,E1 352.413} C_DIS
LIN {X 0.221,Y -467.168,Z 664.751,A 0.000,B 0.000,C 90.000,E1 351.141} C_DIS
LIN {X -0.058,Y -470.573,Z 664.740,A 0.000,B 0.000,C 90.000,E1 349.285} C_DIS
LIN {X 0.144,Y -474.996,Z 664.727,A 0.000,B 0.000,C 90.000,E1 346.756} C_DIS
LIN {X -0.089,Y -477.866,Z 664.718,A 0.000,B 0.000,C 90.000,E1 345.227} C_DIS
LIN {X -0.157,Y -480.790,Z 664.709,A 0.000,B 0.000,C 90.000,E1 343.685} C_DIS
LIN {X -0.035,Y -484.981,Z 664.697,A 0.000,B 0.000,C 90.000,E1 341.511} C_DIS
LIN {X -0.297,Y -488.048,Z 664.689,A 0.000,B 0.000,C 90.000,E1 340.007} C_DIS
LIN {X -0.138,Y -491.725,Z 664.679,A 0.000,B 0.000,C 90.000,E1 338.156} C_DIS
LIN {X 0.061,Y -494.634,Z 664.670,A 0.000,B 0.000,C 90.000,E1 336.613} C_DIS
LIN {X 0.003,Y -496.829,Z 664.663,A 0.000,B 0.000,C 90.000,E1 335.409} C_DIS
LIN {X -0.069,Y -500.551,Z 664.652,A 0.000,B 0.000,C 90.000,E1 333.307} C_DIS
LIN {X -0.042,Y -503.032,Z 664.645,A 0.000,B 0.000,C 90.000,E1 332.103} C_DIS
LIN {X -0.123,Y -504.609,Z 664.642,A 0.000,B 0.000,C 90.000,E1 331.513} C_DIS
LIN {X 0.184,Y -505.503,Z 664.640,A 0.000,B 0.000,C 90.000,E1 331.179} C_DIS
LIN {X 0.063,Y -507.285,Z 664.638,A 0.000,B 0.000,C 90.000,E1 330.745} C_DIS
LIN {X -0.061,Y -508.933,Z 664.636,A 0.000,B 0.000,C 90.000,E1 330.461} C_DIS
LIN {X 0.055,Y -511.183,Z 664.634,A 0.000,B 0.000,C 90.000,E1 330.127} C_DIS
LIN {X -0.127,Y -512.355,Z 664.633,A 0.000,B 0.000,C 90.000,E1 329.999} C_DIS
LIN {X -0.033,Y -515.099,Z 664.632,A 0.000,B 0.000,C 90.000,E1 329.715} C_DIS
LIN {X -0.110,Y -520.341,Z 664.629,A 0.000,B 0.000,C 90.000,E1 329.282} C_DIS
LIN {X -0.326,Y -535.410,Z 664.623,A 0.000,B 0.000,C 90.000,E1 328.201} C_DIS
LIN {X 0.171,Y -542.742,Z 664.620,A 0.000,B 0.000,C 90.000,E1 327.582} C_DIS
LIN {X -0.299,Y -549.856,Z 664.617,A 0.000,B 0.000,C 90.000,E1 327.041} C_DIS
LIN {X -0.215,Y -556.871,Z 664.613,A 0.000,B 0.000,C 90.000,E1 326.421} C_DIS
LIN {X -0.116,Y -563.502,Z 664.610,A 0.000,B 0.000,C 90.000,E1 325.801} C_DIS
LIN {X 0.070,Y -574.144,Z 664.604,A 0.000,B 0.000,C 90.000,E1 324.769} C_DIS
LIN {X 0.050,Y -584.557,Z 664.599,A 0.000,B 0.000,C 90.000,E1 323.749} C_DIS
LIN {X -0.124,Y -590.944,Z 664.595,A 0.000,B 0.000,C 90.000,E1 323.130} C_DIS
LIN {X -0.072,Y -598.448,Z 664.591,A 0.000,B 0.000,C 90.000,E1 322.351} C_DIS
LIN {X 0.000,Y -603.276,Z 664.588,A 0.000,B 0.000,C 90.000,E1 321.823} C_DIS
LIN {X -0.014,Y -609.053,Z 664.584,A 0.000,B 0.000,C 90.000,E1 321.170} C_DIS
LIN {X 0.015,Y -614.495,Z 664.581,A 0.000,B 0.000,C 90.000,E1 320.517} C_DIS
LIN {X -0.384,Y -619.564,Z 664.577,A 0.000,B 0.000,C 90.000,E1 319.908} C_DIS
LIN {X -0.230,Y -623.353,Z 664.574,A 0.000,B 0.000,C 90.000,E1 319.380} C_DIS
LIN {X -0.221,Y -629.582,Z 664.569,A 0.000,B 0.000,C 90.000,E1 318.485} C_DIS
LIN {X 0.315,Y -635.399,Z 664.564,A 0.000,B 0.000,C 90.000,E1 317.553} C_DIS
LIN {X 0.054,Y -640.081,Z 664.560,A 0.000,B 0.000,C 90.000,E1 316.824} C_DIS
LIN {X 0.273,Y -644.645,Z 664.556,A 0.000,B 0.000,C 90.000,E1 316.053} C_DIS
LIN {X -0.007,Y -651.141,Z 664.550,A 0.000,B 0.000,C 90.000,E1 314.960} C_DIS
LIN {X -0.166,Y -656.014,Z 664.545,A 0.000,B 0.000,C 90.000,E1 314.109} C_DIS
LIN {X 0.171,Y -662.296,Z 664.538,A 0.000,B 0.000,C 90.000,E1 312.852} C_DIS
LIN {X 0.147,Y -666.450,Z 664.533,A 0.000,B 0.000,C 90.000,E1 312.000} C_DIS
LIN {X -0.306,Y -671.017,Z 664.528,A 0.000,B 0.000,C 90.000,E1 311.067} C_DIS
LIN {X 0.214,Y -673.163,Z 664.525,A 0.000,B 0.000,C 90.000,E1 310.539} C_DIS
LIN {X 0.350,Y -677.211,Z 664.520,A 0.000,B 0.000,C 90.000,E1 309.564} C_DIS
LIN {X -0.018,Y -679.847,Z 664.516,A 0.000,B 0.000,C 90.000,E1 308.874} C_DIS
LIN {X -0.232,Y -683.102,Z 664.511,A 0.000,B 0.000,C 90.000,E1 307.935} C_DIS
LIN {X -0.019,Y -685.297,Z 664.507,A 0.000,B 0.000,C 90.000,E1 307.202} C_DIS
LIN {X -0.020,Y -687.971,Z 664.501,A 0.000,B 0.000,C 90.000,E1 306.251} C_DIS
LIN {X 0.239,Y -689.872,Z 664.497,A 0.000,B 0.000,C 90.000,E1 305.518} C_DIS
LIN {X -0.249,Y -692.204,Z 664.492,A 0.000,B 0.000,C 90.000,E1 304.612} C_DIS
LIN {X -0.134,Y -694.304,Z 664.487,A 0.000,B 0.000,C 90.000,E1 303.658} C_DIS
LIN {X 0.014,Y -696.208,Z 664.482,A 0.000,B 0.000,C 90.000,E1 302.704} C_DIS
LIN {X 0.188,Y -697.899,Z 664.477,A 0.000,B 0.000,C 90.000,E1 301.750} C_DIS
LIN {X 0.033,Y -699.799,Z 664.470,A 0.000,B 0.000,C 90.000,E1 300.590} C_DIS
LIN {X -0.118,Y -701.050,Z 664.465,A 0.000,B 0.000,C 90.000,E1 299.667} C_DIS
LIN {X -0.044,Y -702.847,Z 664.456,A 0.000,B 0.000,C 90.000,E1 298.025} C_DIS
LIN {X 0.076,Y -704.161,Z 664.448,A 0.000,B 0.000,C 90.000,E1 296.616} C_DIS
LIN {X -0.007,Y -704.699,Z 664.444,A 0.000,B 0.000,C 90.000,E1 295.924} C_DIS
LIN {X -0.354,Y -704.843,Z 664.443,A 0.000,B 0.000,C 90.000,E1 295.720} C_DIS
LIN {X -0.067,Y -704.703,Z 664.441,A 0.000,B 0.000,C 90.000,E1 295.463} C_DIS
LIN {X 0.209,Y -704.128,Z 664.439,A 0.000,B 0.000,C 90.000,E1 294.975} C_DIS
LIN {X -0.143,Y -703.252,Z 664.438,A 0.000,B 0.000,C 90.000,E1 294.771} C_DIS
LIN {X 0.129,Y -700.680,Z 664.435,A 0.000,B 0.000,C 90.000,E1 294.283} C_DIS
LIN {X -0.373,Y -699.778,Z 664.434,A 0.000,B 0.000,C 90.000,E1 294.207} C_DIS
LIN {X -0.236,Y -698.435,Z 664.434,A 0.000,B 0.000,C 90.000,E1 294.079} C_DIS
LIN {X 0.212,Y -691.905,Z 664.432,A 0.000,B 0.000,C 90.000,E1 293.643} C_DIS
LIN {X 0.032,Y -689.777,Z 664.431,A 0.000,B 0.000,C 90.000,E1 293.567} C_DIS
LIN {X 0.121,Y -688.213,Z 664.431,A 0.000,B 0.000,C 90.000,E1 293.515} C_DIS
LIN {X -0.213,Y -680.642,Z 664.430,A 0.000,B 0.000,C 90.000,E1 293.387} C_DIS
LIN {X -0.037,Y -671.952,Z 664.429,A 0.000,B 0.000,C 90.000,E1 293.259} C_DIS
LIN {X -0.131,Y -665.325,Z 664.429,A 0.000,B 0.000,C 90.000,E1 293.206} C_DIS
LIN {X -0.129,Y -652.335,Z 664.428,A 0.000,B 0.000,C 90.000,E1 293.025} C_DIS
LIN {X 0.188,Y -642.631,Z 664.427,A 0.000,B 0.000,C 90.000,E1 292.823} C_DIS
LIN {X -0.170,Y -629.127,Z 664.425,A 0.000,B 0.000,C 90.000,E1 292.567} C_DIS
LIN {X 0.015,Y -615.785,Z 664.423,A 0.000,B 0.000,C 90.000,E1 292.206} C_DIS
LIN {X -0.252,Y -588.562,Z 664.419,A 0.000,B 0.000,C 90.000,E1 291.408} C_DIS
LIN {X 0.006,Y -577.956,Z 664.417,A 0.000,B 0.000,C 90.000,E1 291.046} C_DIS
LIN {X -0.179,Y -563.580,Z 664.415,A 0.000,B 0.000,C 90.000,E1 290.663} C_DIS
LIN {X -0.131,Y -561.110,Z 664.414,A 0.000,B 0.000,C 90.000,E1 290.556} C_DIS
LIN {X 0.023,Y -556.276,Z 664.413,A 0.000,B 0.000,C 90.000,E1 290.301} C_DIS
LIN {X -0.026,Y -556.219,Z 664.413,A 0.000,B 0.000,C 90.000,E1 290.301} C_DIS
LIN {X -0.093,Y -555.318,Z 664.412,A 0.000,B 0.000,C 90.000,E1 290.174} C_DIS
LIN {X -0.135,Y -555.303,Z 664.412,A 0.000,B 0.000,C 90.000,E1 290.174} C_DIS
LIN {X 0.118,Y -554.714,Z 664.410,A 0.000,B 0.000,C 90.000,E1 289.704} C_DIS
LIN {X -0.257,Y -554.467,Z 664.405,A 0.000,B 0.000,C 90.000,E1 288.906} C_DIS
LIN {X -0.008,Y -554.326,Z 664.399,A 0.000,B 0.000,C 90.000,E1 287.764} C_DIS
LIN {X -0.174,Y -553.947,Z 664.391,A 0.000,B 0.000,C 90.000,E1 286.386} C_DIS
LIN {X -0.236,Y -553.356,Z 664.382,A 0.000,B 0.000,C 90.000,E1 284.717} C_DIS
LIN {X -0.157,Y -552.758,Z 664.375,A 0.000,B 0.000,C 90.000,E1 283.592} C_DIS
LIN {X 0.255,Y -551.745,Z 664.365,A 0.000,B 0.000,C 90.000,E1 281.591} C_DIS
LIN {X -0.012,Y -550.735,Z 664.352,A 0.000,B 0.000,C 90.000,E1 279.378} C_DIS
LIN {X -0.065,Y -550.238,Z 664.343,A 0.000,B 0.000,C 90.000,E1 277.701} C_DIS
LIN {X -0.131,Y -549.887,Z 664.333,A 0.000,B 0.000,C 90.000,E1 276.024} C_DIS
LIN {X -0.182,Y -549.623,Z 664.321,A 0.000,B 0.000,C 90.000,E1 273.784} C_DIS
LIN {X 0.050,Y -549.389,Z 664.315,A 0.000,B 0.000,C 90.000,E1 272.636} C_DIS
LIN {X 0.275,Y -549.076,Z 664.308,A 0.000,B 0.000,C 90.000,E1 271.489} C_DIS
LIN {X -0.016,Y -548.448,Z 664.301,A 0.000,B 0.000,C 90.000,E1 270.115} C_DIS
LIN {X 0.231,Y -547.708,Z 664.293,A 0.000,B 0.000,C 90.000,E1 268.682} C_DIS
LIN {X -0.115,Y -547.085,Z 664.287,A 0.000,B 0.000,C 90.000,E1 267.593} C_DIS
LIN {X 0.118,Y -546.283,Z 664.279,A 0.000,B 0.000,C 90.000,E1 266.159} C_DIS
LIN {X -0.176,Y -545.209,Z 664.271,A 0.000,B 0.000,C 90.000,E1 264.780} C_DIS
LIN {X 0.109,Y -544.015,Z 664.263,A 0.000,B 0.000,C 90.000,E1 263.337} C_DIS
LIN {X -0.085,Y -541.964,Z 664.252,A 0.000,B 0.000,C 90.000,E1 261.376} C_DIS
LIN {X 0.044,Y -539.210,Z 664.236,A 0.000,B 0.000,C 90.000,E1 258.522} C_DIS
LIN {X 0.113,Y -537.521,Z 664.225,A 0.000,B 0.000,C 90.000,E1 256.520} C_DIS
LIN {X 0.025,Y -536.325,Z 664.217,A 0.000,B 0.000,C 90.000,E1 255.102} C_DIS
LIN {X -0.138,Y -535.289,Z 664.211,A 0.000,B 0.000,C 90.000,E1 253.976} C_DIS
LIN {X 0.065,Y -533.535,Z 664.201,A 0.000,B 0.000,C 90.000,E1 252.236} C_DIS
LIN {X 0.204,Y -532.158,Z 664.193,A 0.000,B 0.000,C 90.000,E1 250.786} C_DIS
LIN {X 0.117,Y -530.845,Z 664.187,A 0.000,B 0.000,C 90.000,E1 249.645} C_DIS
LIN {X 0.059,Y -528.435,Z 664.177,A 0.000,B 0.000,C 90.000,E1 247.922} C_DIS
LIN {X -0.022,Y -526.388,Z 664.169,A 0.000,B 0.000,C 90.000,E1 246.485} C_DIS
LIN {X -0.140,Y -523.850,Z 664.161,A 0.000,B 0.000,C 90.000,E1 245.049} C_DIS
LIN {X -0.237,Y -521.792,Z 664.155,A 0.000,B 0.000,C 90.000,E1 243.896} C_DIS
LIN {X 0.014,Y -518.875,Z 664.147,A 0.000,B 0.000,C 90.000,E1 242.410} C_DIS
LIN {X 0.209,Y -515.863,Z 664.139,A 0.000,B 0.000,C 90.000,E1 240.923} C_DIS
LIN {X 0.147,Y -512.664,Z 664.130,A 0.000,B 0.000,C 90.000,E1 239.459} C_DIS
